LIN {X 0,Y 394.141,Z 720.215,A -85,B 0,C 180,E1 -9307.32,E2 -9307.32} C_VEL
LIN {X 0,Y 395.214,Z 710.247,A -85,B 0,C 180,E1 -9309.27,E2 -9309.27} C_VEL
LIN {X 0,Y 396.4,Z 699.307,A -85,B 0,C 180,E1 -9310.978,E2 -9310.978} C_VEL
LIN {X 0,Y 397.775,Z 685.884,A -85,B 0,C 180,E1 -9312.64,E2 -9312.64} C_VEL
LIN {X 0,Y 399.025,Z 672.379,A -85,B 0,C 180,E1 -9313.952,E2 -9313.952} C_VEL
LIN {X 0,Y 400.251,Z 656.946,A -85,B 0,C 180,E1 -9315.107,E2 -9315.107} C_VEL
LIN {X 0,Y 401.169,Z 641.449,A -85,B 0,C 180,E1 -9315.955,E2 -9315.955} C_VEL
LIN {X 0,Y 401.832,Z 624.77,A -85,B 0,C 180,E1 -9316.577,E2 -9316.577} C_VEL
LIN {X 0,Y 402.409,Z 593.858,A -85,B 0,C 180,E1 -9317.193,E2 -9317.193} C_VEL
LIN {X 0,Y 404.148,Z 493.038,A -85,B 0,C 180,E1 -9319.051,E2 -9319.051} C_VEL
LIN {X 0,Y 402.544,Z 478.977,A -85,B 0,C 180,E1 -9319.466,E2 -9319.466} C_VEL
LIN {X 0,Y 404.689,Z 437.04,A -85,B 0,C 180,E1 -9323.279,E2 -9323.279} C_VEL
LIN {X 0,Y 407.087,Z 392.855,A -85,B 0,C 180,E1 -9327.292,E2 -9327.292} C_VEL
LIN {X 0,Y 409.144,Z 348.932,A -85,B 0,C 180,E1 -9331.221,E2 -9331.221} C_VEL
LIN {X 0,Y 409.823,Z 331.006,A -85,B 0,C 180,E1 -9332.855,E2 -9332.855} C_VEL
LIN {X 0,Y 403.97,Z 313.246,A -85,B 0,C 180,E1 -9335.117,E2 -9335.117} C_VEL
LIN {X 0,Y 396.828,Z 295.284,A -85,B 0,C 180,E1 -9337.637,E2 -9337.637} C_VEL
LIN {X 0,Y 393.6,Z 287.76,A -85,B 0,C 180,E1 -9338.814,E2 -9338.814} C_VEL
LIN {X 0,Y 393.563,Z 287.458,A -85,B 0,C 180,E1 -9340.56,E2 -9340.56} C_VEL
LIN {X 0,Y 393.566,Z 287.451,A -85,B 0,C 180,E1 -9344.528,E2 -9344.528} C_VEL
LIN {X 0,Y 393.561,Z 287.464,A -85,B 0,C 180,E1 -9348.57,E2 -9348.57} C_VEL
LIN {X 0,Y 393.57,Z 287.463,A -85,B 0,C 180,E1 -9352.555,E2 -9352.555} C_VEL
LIN {X 0,Y 393.561,Z 287.461,A -85,B 0,C 180,E1 -9356.65,E2 -9356.65} C_VEL
LIN {X 0,Y 393.569,Z 287.456,A -85,B 0,C 180,E1 -9360.727,E2 -9360.727} C_VEL
LIN {X 0,Y 393.564,Z 287.462,A -85,B 0,C 180,E1 -9364.809,E2 -9364.809} C_VEL
LIN {X 0,Y 393.566,Z 287.458,A -85,B 0,C 180,E1 -9368.804,E2 -9368.804} C_VEL
LIN {X 0,Y 393.564,Z 287.456,A -85,B 0,C 180,E1 -9372.769,E2 -9372.769} C_VEL
LIN {X 0,Y 393.562,Z 287.46,A -85,B 0,C 180,E1 -9376.716,E2 -9376.716} C_VEL
LIN {X 0,Y 393.566,Z 287.46,A -85,B 0,C 180,E1 -9380.793,E2 -9380.793} C_VEL
LIN {X 0,Y 393.562,Z 287.459,A -85,B 0,C 180,E1 -9384.783,E2 -9384.783} C_VEL
LIN {X 0,Y 393.572,Z 287.46,A -85,B 0,C 180,E1 -9388.861,E2 -9388.861} C_VEL
LIN {X 0,Y 393.559,Z 287.463,A -85,B 0,C 180,E1 -9392.766,E2 -9392.766} C_VEL
LIN {X 0,Y 393.553,Z 287.462,A -85,B 0,C 180,E1 -9396.658,E2 -9396.658} C_VEL
LIN {X 0,Y 393.55,Z 287.466,A -85,B 0,C 180,E1 -9400.571,E2 -9400.571} C_VEL
LIN {X 0,Y 393.582,Z 287.73,A -85,B 0,C 180,E1 -9402.449,E2 -9402.449} C_VEL
LIN {X 0,Y 402.202,Z 308.042,A -85,B 0,C 180,E1 -9405.925,E2 -9405.925} C_VEL
LIN {X 0,Y 406.944,Z 319.226,A -85,B 0,C 180,E1 -9407.641,E2 -9407.641} C_VEL
LIN {X 0,Y 422.36,Z 346.857,A -85,B 0,C 180,E1 -9409.922,E2 -9409.922} C_VEL
LIN {X 0,Y 422.986,Z 349.882,A -85,B 0,C 180,E1 -9410.056,E2 -9410.056} C_VEL
LIN {X 0,Y 415.677,Z 539.395,A -85,B 0,C 180,E1 -9413.938,E2 -9413.938} C_VEL
LIN {X 0,Y 414.165,Z 578.769,A -85,B 0,C 180,E1 -9414.777,E2 -9414.777} C_VEL
LIN {X 0,Y 412.749,Z 599.725,A -85,B 0,C 180,E1 -9415.461,E2 -9415.461} C_VEL
LIN {X 0,Y 410.909,Z 620.31,A -85,B 0,C 180,E1 -9416.39,E2 -9416.39} C_VEL
LIN {X 0,Y 408.749,Z 640.92,A -85,B 0,C 180,E1 -9417.61,E2 -9417.61} C_VEL
LIN {X 0,Y 406.395,Z 660.376,A -85,B 0,C 180,E1 -9419.058,E2 -9419.058} C_VEL
LIN {X 0,Y 403.973,Z 678.786,A -85,B 0,C 180,E1 -9420.739,E2 -9420.739} C_VEL
LIN {X 0,Y 401.555,Z 696.152,A -85,B 0,C 180,E1 -9422.654,E2 -9422.654} C_VEL
LIN {X 0,Y 399.377,Z 711.376,A -85,B 0,C 180,E1 -9424.659,E2 -9424.659} C_VEL
LIN {X 0,Y 397.371,Z 725.681,A -85,B 0,C 180,E1 -9426.89,E2 -9426.89} C_VEL
LIN {X 0,Y 395.647,Z 738.602,A -85,B 0,C 180,E1 -9429.282,E2 -9429.282} C_VEL
LIN {X 0,Y 394.254,Z 750.119,A -85,B 0,C 180,E1 -9431.826,E2 -9431.826} C_VEL
LIN {X 0,Y 393.264,Z 759.694,A -85,B 0,C 180,E1 -9434.367,E2 -9434.367} C_VEL
LIN {X 0,Y 392.539,Z 768.289,A -85,B 0,C 180,E1 -9437.199,E2 -9437.199} C_VEL
LIN {X 0,Y 392.165,Z 774.955,A -85,B 0,C 180,E1 -9440.018,E2 -9440.018} C_VEL
LIN {X 0,Y 392.007,Z 779.883,A -85,B 0,C 180,E1 -9442.831,E2 -9442.831} C_VEL
LIN {X 0,Y 391.988,Z 783.143,A -85,B 0,C 180,E1 -9445.613,E2 -9445.613} C_VEL
LIN {X 0,Y 391.999,Z 784.826,A -85,B 0,C 180,E1 -9448.394,E2 -9448.394} C_VEL
LIN {X 0,Y 392.011,Z 784.855,A -85,B 0,C 180,E1 -9451.072,E2 -9451.072} C_VEL
LIN {X 0,Y 392.001,Z 783.287,A -85,B 0,C 180,E1 -9453.95,E2 -9453.95} C_VEL
LIN {X 0,Y 392.02,Z 780.159,A -85,B 0,C 180,E1 -9456.739,E2 -9456.739} C_VEL
LIN {X 0,Y 392.132,Z 775.337,A -85,B 0,C 180,E1 -9459.542,E2 -9459.542} C_VEL
LIN {X 0,Y 392.433,Z 769.064,A -85,B 0,C 180,E1 -9462.21,E2 -9462.21} C_VEL
LIN {X 0,Y 393.049,Z 760.59,A -85,B 0,C 180,E1 -9465.04,E2 -9465.04} C_VEL
LIN {X 0,Y 393.982,Z 750.577,A -85,B 0,C 180,E1 -9467.732,E2 -9467.732} C_VEL
LIN {X 0,Y 395.262,Z 739.097,A -85,B 0,C 180,E1 -9470.278,E2 -9470.278} C_VEL
LIN {X 0,Y 396.852,Z 726.19,A -85,B 0,C 180,E1 -9472.675,E2 -9472.675} C_VEL
LIN {X 0,Y 398.795,Z 711.301,A -85,B 0,C 180,E1 -9474.992,E2 -9474.992} C_VEL
LIN {X 0,Y 401.008,Z 694.704,A -85,B 0,C 180,E1 -9477.149,E2 -9477.149} C_VEL
LIN {X 0,Y 403.385,Z 676.518,A -85,B 0,C 180,E1 -9479.116,E2 -9479.116} C_VEL
LIN {X 0,Y 405.775,Z 657.251,A -85,B 0,C 180,E1 -9480.834,E2 -9480.834} C_VEL
LIN {X 0,Y 408.122,Z 636.959,A -85,B 0,C 180,E1 -9482.306,E2 -9482.306} C_VEL
LIN {X 0,Y 410.253,Z 616.233,A -85,B 0,C 180,E1 -9483.507,E2 -9483.507} C_VEL
LIN {X 0,Y 412.2,Z 594.587,A -85,B 0,C 180,E1 -9484.469,E2 -9484.469} C_VEL
LIN {X 0,Y 413.812,Z 572.25,A -85,B 0,C 180,E1 -9485.184,E2 -9485.184} C_VEL
LIN {X 0,Y 418.128,Z 493.872,A -85,B 0,C 180,E1 -9487.09,E2 -9487.09} C_VEL
LIN {X 0,Y 423.367,Z 428.006,A -85,B 0,C 180,E1 -9488.865,E2 -9488.865} C_VEL
LIN {X 0,Y 430.317,Z 363.895,A -85,B 0,C 180,E1 -9490.73,E2 -9490.73} C_VEL
LIN {X 0,Y 431.806,Z 351.842,A -85,B 0,C 180,E1 -9491.098,E2 -9491.098} C_VEL
LIN {X 0,Y 429.203,Z 345.73,A -85,B 0,C 180,E1 -9492.25,E2 -9492.25} C_VEL
LIN {X 0,Y 426.845,Z 341.145,A -85,B 0,C 180,E1 -9493.567,E2 -9493.567} C_VEL
LIN {X 0,Y 424.814,Z 337.789,A -85,B 0,C 180,E1 -9495.493,E2 -9495.493} C_VEL
LIN {X 0,Y 424.298,Z 337.772,A -85,B 0,C 180,E1 -9496.734,E2 -9496.734} C_VEL
LIN {X 0,Y 424.813,Z 340.3,A -85,B 0,C 180,E1 -9498.662,E2 -9498.662} C_VEL
LIN {X 0,Y 426.33,Z 344.624,A -85,B 0,C 180,E1 -9500.189,E2 -9500.189} C_VEL
LIN {X 0,Y 428.359,Z 350.001,A -85,B 0,C 180,E1 -9501.494,E2 -9501.494} C_VEL
LIN {X 0,Y 429.496,Z 353.537,A -85,B 0,C 180,E1 -9502.122,E2 -9502.122} C_VEL
LIN {X 0,Y 429.664,Z 372.072,A -85,B 0,C 180,E1 -9503.417,E2 -9503.417} C_VEL
LIN {X 0,Y 429.502,Z 378.771,A -85,B 0,C 180,E1 -9503.782,E2 -9503.782} C_VEL
LIN {X 0,Y 420.852,Z 453.997,A -85,B 0,C 180,E1 -9506.036,E2 -9506.036} C_VEL
LIN {X 0,Y 414.952,Z 523.412,A -85,B 0,C 180,E1 -9508.016,E2 -9508.016} C_VEL
LIN {X 0,Y 411.775,Z 569.755,A -85,B 0,C 180,E1 -9509.309,E2 -9509.309} C_VEL
LIN {X 0,Y 410.048,Z 589.973,A -85,B 0,C 180,E1 -9510.13,E2 -9510.13} C_VEL
LIN {X 0,Y 408.054,Z 609.913,A -85,B 0,C 180,E1 -9511.208,E2 -9511.208} C_VEL
LIN {X 0,Y 405.951,Z 628.582,A -85,B 0,C 180,E1 -9512.496,E2 -9512.496} C_VEL
LIN {X 0,Y 403.72,Z 646.478,A -85,B 0,C 180,E1 -9514.03,E2 -9514.03} C_VEL
LIN {X 0,Y 401.544,Z 662.795,A -85,B 0,C 180,E1 -9515.742,E2 -9515.742} C_VEL
LIN {X 0,Y 399.466,Z 677.763,A -85,B 0,C 180,E1 -9517.639,E2 -9517.639} C_VEL
LIN {X 0,Y 397.58,Z 691.237,A -85,B 0,C 180,E1 -9519.693,E2 -9519.693} C_VEL
LIN {X 0,Y 395.933,Z 703.264,A -85,B 0,C 180,E1 -9521.904,E2 -9521.904} C_VEL
LIN {X 0,Y 394.567,Z 713.847,A -85,B 0,C 180,E1 -9524.268,E2 -9524.268} C_VEL
LIN {X 0,Y 393.512,Z 722.946,A -85,B 0,C 180,E1 -9526.781,E2 -9526.781} C_VEL
LIN {X 0,Y 392.803,Z 730.143,A -85,B 0,C 180,E1 -9529.292,E2 -9529.292} C_VEL
LIN {X 0,Y 392.356,Z 735.897,A -85,B 0,C 180,E1 -9531.943,E2 -9531.943} C_VEL
LIN {X 0,Y 392.136,Z 739.907,A -85,B 0,C 180,E1 -9534.587,E2 -9534.587} C_VEL
LIN {X 0,Y 392.039,Z 742.339,A -85,B 0,C 180,E1 -9537.369,E2 -9537.369} C_VEL
LIN {X 0,Y 392.022,Z 743.022,A -85,B 0,C 180,E1 -9540.001,E2 -9540.001} C_VEL
LIN {X 0,Y 392.027,Z 742.021,A -85,B 0,C 180,E1 -9542.778,E2 -9542.778} C_VEL
LIN {X 0,Y 392.1,Z 739.253,A -85,B 0,C 180,E1 -9545.561,E2 -9545.561} C_VEL
LIN {X 0,Y 392.314,Z 734.637,A -85,B 0,C 180,E1 -9548.354,E2 -9548.354} C_VEL
LIN {X 0,Y 392.742,Z 728.456,A -85,B 0,C 180,E1 -9551.008,E2 -9551.008} C_VEL
LIN {X 0,Y 393.485,Z 720.325,A -85,B 0,C 180,E1 -9553.67,E2 -9553.67} C_VEL
LIN {X 0,Y 394.55,Z 710.631,A -85,B 0,C 180,E1 -9556.187,E2 -9556.187} C_VEL
LIN {X 0,Y 395.927,Z 699.422,A -85,B 0,C 180,E1 -9558.554,E2 -9558.554} C_VEL
LIN {X 0,Y 397.59,Z 686.704,A -85,B 0,C 180,E1 -9560.769,E2 -9560.769} C_VEL
LIN {X 0,Y 399.492,Z 672.419,A -85,B 0,C 180,E1 -9562.827,E2 -9562.827} C_VEL
LIN {X 0,Y 401.465,Z 657.392,A -85,B 0,C 180,E1 -9564.625,E2 -9564.625} C_VEL
LIN {X 0,Y 403.508,Z 640.935,A -85,B 0,C 180,E1 -9566.252,E2 -9566.252} C_VEL
LIN {X 0,Y 405.56,Z 622.985,A -85,B 0,C 180,E1 -9567.693,E2 -9567.693} C_VEL
LIN {X 0,Y 407.476,Z 603.872,A -85,B 0,C 180,E1 -9568.908,E2 -9568.908} C_VEL
LIN {X 0,Y 409.102,Z 584.185,A -85,B 0,C 180,E1 -9569.862,E2 -9569.862} C_VEL
LIN {X 0,Y 410.384,Z 564.626,A -85,B 0,C 180,E1 -9570.537,E2 -9570.537} C_VEL
LIN {X 0,Y 411.678,Z 531.02,A -85,B 0,C 180,E1 -9571.28,E2 -9571.28} C_VEL
LIN {X 0,Y 417.674,Z 373.67,A -85,B 0,C 180,E1 -9574.608,E2 -9574.608} C_VEL
LIN {X 0,Y 412.809,Z 339.814,A -85,B 0,C 180,E1 -9575.949,E2 -9575.949} C_VEL
LIN {X 0,Y 412.541,Z 337.856,A -85,B 0,C 180,E1 -9576.187,E2 -9576.187} C_VEL
LIN {X 0,Y 406.059,Z 319.468,A -85,B 0,C 180,E1 -9579.024,E2 -9579.024} C_VEL
LIN {X 0,Y 398.94,Z 301.069,A -85,B 0,C 180,E1 -9582.108,E2 -9582.108} C_VEL
LIN {X 0,Y 393.582,Z 287.659,A -85,B 0,C 180,E1 -9584.556,E2 -9584.556} C_VEL
LIN {X 0,Y 393.563,Z 287.462,A -85,B 0,C 180,E1 -9588.544,E2 -9588.544} C_VEL
LIN {X 0,Y 393.56,Z 287.462,A -85,B 0,C 180,E1 -9592.435,E2 -9592.435} C_VEL
LIN {X 0,Y 393.564,Z 287.463,A -85,B 0,C 180,E1 -9596.44,E2 -9596.44} C_VEL
LIN {X 0,Y 393.559,Z 287.441,A -85,B 0,C 180,E1 -9600.469,E2 -9600.469} C_VEL
LIN {X 0,Y 393.552,Z 287.446,A -85,B 0,C 180,E1 -9604.412,E2 -9604.412} C_VEL
LIN {X 0,Y 393.548,Z 287.449,A -85,B 0,C 180,E1 -9608.382,E2 -9608.382} C_VEL
LIN {X 0,Y 393.536,Z 287.554,A -85,B 0,C 180,E1 -9611.174,E2 -9611.174} C_VEL
LIN {X 0,Y 393.987,Z 289.28,A -85,B 0,C 180,E1 -9611.503,E2 -9611.503} C_VEL
LIN {X 0,Y 401.135,Z 306.789,A -85,B 0,C 180,E1 -9614.011,E2 -9614.011} C_VEL
LIN {X 0,Y 407.641,Z 325.401,A -85,B 0,C 180,E1 -9616.467,E2 -9616.467} C_VEL
LIN {X 0,Y 407.824,Z 328.938,A -85,B 0,C 180,E1 -9616.828,E2 -9616.828} C_VEL
LIN {X 0,Y 406.05,Z 334.761,A -85,B 0,C 180,E1 -9617.234,E2 -9617.234} C_VEL
LIN {X 0,Y 402.635,Z 343.48,A -85,B 0,C 180,E1 -9617.778,E2 -9617.778} C_VEL
LIN {X 0,Y 402.207,Z 346.122,A -85,B 0,C 180,E1 -9617.999,E2 -9617.999} C_VEL
LIN {X 0,Y 399.838,Z 387.755,A -85,B 0,C 180,E1 -9621.876,E2 -9621.876} C_VEL
LIN {X 0,Y 397.374,Z 430.242,A -85,B 0,C 180,E1 -9625.814,E2 -9625.814} C_VEL
LIN {X 0,Y 394.991,Z 472.14,A -85,B 0,C 180,E1 -9629.708,E2 -9629.708} C_VEL
LIN {X 0,Y 394.7,Z 479.497,A -85,B 0,C 180,E1 -9630.357,E2 -9630.357} C_VEL
LIN {X 0,Y 396.483,Z 496.869,A -85,B 0,C 180,E1 -9630.818,E2 -9630.818} C_VEL
LIN {X 0,Y 394.065,Z 622.743,A -85,B 0,C 180,E1 -9633.176,E2 -9633.176} C_VEL
LIN {X 0,Y 393.45,Z 638.836,A -85,B 0,C 180,E1 -9633.746,E2 -9633.746} C_VEL
LIN {X 0,Y 392.507,Z 654.948,A -85,B 0,C 180,E1 -9634.601,E2 -9634.601} C_VEL
LIN {X 0,Y 391.39,Z 669.303,A -85,B 0,C 180,E1 -9635.643,E2 -9635.643} C_VEL
LIN {X 0,Y 390.069,Z 683.635,A -85,B 0,C 180,E1 -9636.992,E2 -9636.992} C_VEL
LIN {X 0,Y 388.772,Z 696.257,A -85,B 0,C 180,E1 -9638.502,E2 -9638.502} C_VEL
LIN {X 0,Y 387.5,Z 707.934,A -85,B 0,C 180,E1 -9640.254,E2 -9640.254} C_VEL
LIN {X 0,Y 386.423,Z 717.792,A -85,B 0,C 180,E1 -9642.096,E2 -9642.096} C_VEL
LIN {X 0,Y 385.467,Z 726.899,A -85,B 0,C 180,E1 -9644.264,E2 -9644.264} C_VEL
LIN {X 0,Y 384.8,Z 734.119,A -85,B 0,C 180,E1 -9646.5,E2 -9646.5} C_VEL
LIN {X 0,Y 384.362,Z 739.874,A -85,B 0,C 180,E1 -9648.974,E2 -9648.974} C_VEL
LIN {X 0,Y 384.158,Z 743.496,A -85,B 0,C 180,E1 -9651.368,E2 -9651.368} C_VEL
LIN {X 0,Y 384.083,Z 745.361,A -85,B 0,C 180,E1 -9653.795,E2 -9653.795} C_VEL
LIN {X 0,Y 384.087,Z 745.527,A -85,B 0,C 180,E1 -9656.098,E2 -9656.098} C_VEL
LIN {X 0,Y 384.166,Z 743.839,A -85,B 0,C 180,E1 -9658.611,E2 -9658.611} C_VEL
LIN {X 0,Y 384.38,Z 740.5,A -85,B 0,C 180,E1 -9660.998,E2 -9660.998} C_VEL
LIN {X 0,Y 384.766,Z 735.571,A -85,B 0,C 180,E1 -9663.249,E2 -9663.249} C_VEL
LIN {X 0,Y 385.43,Z 728.74,A -85,B 0,C 180,E1 -9665.524,E2 -9665.524} C_VEL
LIN {X 0,Y 386.342,Z 720.344,A -85,B 0,C 180,E1 -9667.643,E2 -9667.643} C_VEL
LIN {X 0,Y 387.506,Z 710.223,A -85,B 0,C 180,E1 -9669.649,E2 -9669.649} C_VEL
LIN {X 0,Y 388.761,Z 699.273,A -85,B 0,C 180,E1 -9671.372,E2 -9671.372} C_VEL
LIN {X 0,Y 390.138,Z 686.536,A -85,B 0,C 180,E1 -9672.975,E2 -9672.975} C_VEL
LIN {X 0,Y 391.426,Z 673.431,A -85,B 0,C 180,E1 -9674.284,E2 -9674.284} C_VEL
LIN {X 0,Y 392.715,Z 658.035,A -85,B 0,C 180,E1 -9675.467,E2 -9675.467} C_VEL
LIN {X 0,Y 393.695,Z 642.674,A -85,B 0,C 180,E1 -9676.34,E2 -9676.34} C_VEL
LIN {X 0,Y 394.411,Z 625.713,A -85,B 0,C 180,E1 -9676.993,E2 -9676.993} C_VEL
LIN {X 0,Y 394.914,Z 601.292,A -85,B 0,C 180,E1 -9677.508,E2 -9677.508} C_VEL
LIN {X 0,Y 396.897,Z 494.063,A -85,B 0,C 180,E1 -9679.516,E2 -9679.516} C_VEL
LIN {X 0,Y 395.229,Z 479.296,A -85,B 0,C 180,E1 -9679.968,E2 -9679.968} C_VEL
LIN {X 0,Y 397.566,Z 436.543,A -85,B 0,C 180,E1 -9683.895,E2 -9683.895} C_VEL
LIN {X 0,Y 399.816,Z 396.458,A -85,B 0,C 180,E1 -9687.559,E2 -9687.559} C_VEL
LIN {X 0,Y 401.861,Z 357.064,A -85,B 0,C 180,E1 -9691.138,E2 -9691.138} C_VEL
LIN {X 0,Y 402.887,Z 334.115,A -85,B 0,C 180,E1 -9693.228,E2 -9693.228} C_VEL
LIN {X 0,Y 397.283,Z 316.981,A -85,B 0,C 180,E1 -9695.464,E2 -9695.464} C_VEL
LIN {X 0,Y 390.583,Z 299.994,A -85,B 0,C 180,E1 -9697.894,E2 -9697.894} C_VEL
LIN {X 0,Y 386.577,Z 291.412,A -85,B 0,C 180,E1 -9699.246,E2 -9699.246} C_VEL
LIN {X 0,Y 385.632,Z 288.744,A -85,B 0,C 180,E1 -9699.709,E2 -9699.709} C_VEL
LIN {X 0,Y 385.591,Z 288.444,A -85,B 0,C 180,E1 -9701.713,E2 -9701.713} C_VEL
LIN {X 0,Y 385.59,Z 288.452,A -85,B 0,C 180,E1 -9705.738,E2 -9705.738} C_VEL
LIN {X 0,Y 385.591,Z 288.453,A -85,B 0,C 180,E1 -9709.693,E2 -9709.693} C_VEL
LIN {X 0,Y 385.59,Z 288.45,A -85,B 0,C 180,E1 -9713.747,E2 -9713.747} C_VEL
LIN {X 0,Y 385.59,Z 288.455,A -85,B 0,C 180,E1 -9717.77,E2 -9717.77} C_VEL
LIN {X 0,Y 385.591,Z 288.45,A -85,B 0,C 180,E1 -9721.783,E2 -9721.783} C_VEL
LIN {X 0,Y 385.592,Z 288.454,A -85,B 0,C 180,E1 -9725.804,E2 -9725.804} C_VEL
LIN {X 0,Y 385.593,Z 288.446,A -85,B 0,C 180,E1 -9729.854,E2 -9729.854} C_VEL
LIN {X 0,Y 385.594,Z 288.452,A -85,B 0,C 180,E1 -9733.954,E2 -9733.954} C_VEL
LIN {X 0,Y 385.596,Z 288.453,A -85,B 0,C 180,E1 -9737.973,E2 -9737.973} C_VEL
LIN {X 0,Y 385.593,Z 288.447,A -85,B 0,C 180,E1 -9741.925,E2 -9741.925} C_VEL
LIN {X 0,Y 385.597,Z 288.453,A -85,B 0,C 180,E1 -9745.99,E2 -9745.99} C_VEL
LIN {X 0,Y 385.6,Z 288.449,A -85,B 0,C 180,E1 -9750.029,E2 -9750.029} C_VEL
LIN {X 0,Y 385.6,Z 288.45,A -85,B 0,C 180,E1 -9754.061,E2 -9754.061} C_VEL
LIN {X 0,Y 385.601,Z 288.45,A -85,B 0,C 180,E1 -9758.106,E2 -9758.106} C_VEL
LIN {X 0,Y 385.659,Z 288.721,A -85,B 0,C 180,E1 -9761.528,E2 -9761.528} C_VEL
LIN {X 0,Y 388.596,Z 295.735,A -85,B 0,C 180,E1 -9762.839,E2 -9762.839} C_VEL
LIN {X 0,Y 397.618,Z 316.933,A -85,B 0,C 180,E1 -9766.403,E2 -9766.403} C_VEL
LIN {X 0,Y 398.948,Z 319.876,A -85,B 0,C 180,E1 -9766.802,E2 -9766.802} C_VEL
LIN {X 0,Y 414.538,Z 347.5,A -85,B 0,C 180,E1 -9769.179,E2 -9769.179} C_VEL
LIN {X 0,Y 416.358,Z 351.397,A -85,B 0,C 180,E1 -9769.461,E2 -9769.461} C_VEL
LIN {X 0,Y 408.437,Z 546.701,A -85,B 0,C 180,E1 -9773.542,E2 -9773.542} C_VEL
LIN {X 0,Y 407.015,Z 580.064,A -85,B 0,C 180,E1 -9774.29,E2 -9774.29} C_VEL
LIN {X 0,Y 405.492,Z 601.047,A -85,B 0,C 180,E1 -9775.006,E2 -9775.006} C_VEL
LIN {X 0,Y 403.586,Z 621.322,A -85,B 0,C 180,E1 -9775.953,E2 -9775.953} C_VEL
LIN {X 0,Y 401.48,Z 640.647,A -85,B 0,C 180,E1 -9777.12,E2 -9777.12} C_VEL
LIN {X 0,Y 399.03,Z 660.122,A -85,B 0,C 180,E1 -9778.59,E2 -9778.59} C_VEL
LIN {X 0,Y 396.51,Z 678.559,A -85,B 0,C 180,E1 -9780.299,E2 -9780.299} C_VEL
LIN {X 0,Y 394.072,Z 695.297,A -85,B 0,C 180,E1 -9782.172,E2 -9782.172} C_VEL
LIN {X 0,Y 391.716,Z 711.133,A -85,B 0,C 180,E1 -9784.285,E2 -9784.285} C_VEL
LIN {X 0,Y 389.616,Z 725.484,A -85,B 0,C 180,E1 -9786.563,E2 -9786.563} C_VEL
LIN {X 0,Y 387.808,Z 738.415,A -85,B 0,C 180,E1 -9789.002,E2 -9789.002} C_VEL
LIN {X 0,Y 386.351,Z 749.923,A -85,B 0,C 180,E1 -9791.597,E2 -9791.597} C_VEL
LIN {X 0,Y 385.269,Z 759.915,A -85,B 0,C 180,E1 -9794.327,E2 -9794.327} C_VEL
LIN {X 0,Y 384.53,Z 768.479,A -85,B 0,C 180,E1 -9797.233,E2 -9797.233} C_VEL
LIN {X 0,Y 384.157,Z 775.03,A -85,B 0,C 180,E1 -9800.11,E2 -9800.11} C_VEL
LIN {X 0,Y 384.012,Z 779.583,A -85,B 0,C 180,E1 -9802.822,E2 -9802.822} C_VEL
LIN {X 0,Y 383.999,Z 782.86,A -85,B 0,C 180,E1 -9805.751,E2 -9805.751} C_VEL
LIN {X 0,Y 384.011,Z 784.423,A -85,B 0,C 180,E1 -9808.51,E2 -9808.51} C_VEL
LIN {X 0,Y 384.02,Z 784.396,A -85,B 0,C 180,E1 -9811.195,E2 -9811.195} C_VEL
LIN {X 0,Y 384.009,Z 782.846,A -85,B 0,C 180,E1 -9814.033,E2 -9814.033} C_VEL
LIN {X 0,Y 384.024,Z 779.703,A -85,B 0,C 180,E1 -9816.88,E2 -9816.88} C_VEL
LIN {X 0,Y 384.151,Z 774.855,A -85,B 0,C 180,E1 -9819.742,E2 -9819.742} C_VEL
LIN {X 0,Y 384.471,Z 768.554,A -85,B 0,C 180,E1 -9822.467,E2 -9822.467} C_VEL
LIN {X 0,Y 385.142,Z 760.046,A -85,B 0,C 180,E1 -9825.357,E2 -9825.357} C_VEL
LIN {X 0,Y 386.17,Z 749.788,A -85,B 0,C 180,E1 -9828.155,E2 -9828.155} C_VEL
LIN {X 0,Y 387.524,Z 738.476,A -85,B 0,C 180,E1 -9830.702,E2 -9830.702} C_VEL
LIN {X 0,Y 389.231,Z 725.53,A -85,B 0,C 180,E1 -9833.144,E2 -9833.144} C_VEL
LIN {X 0,Y 391.309,Z 710.607,A -85,B 0,C 180,E1 -9835.504,E2 -9835.504} C_VEL
LIN {X 0,Y 393.671,Z 693.985,A -85,B 0,C 180,E1 -9837.698,E2 -9837.698} C_VEL
LIN {X 0,Y 396.149,Z 676.253,A -85,B 0,C 180,E1 -9839.651,E2 -9839.651} C_VEL
LIN {X 0,Y 398.765,Z 656.587,A -85,B 0,C 180,E1 -9841.437,E2 -9841.437} C_VEL
LIN {X 0,Y 401.223,Z 636.704,A -85,B 0,C 180,E1 -9842.907,E2 -9842.907} C_VEL
LIN {X 0,Y 403.581,Z 615.51,A -85,B 0,C 180,E1 -9844.16,E2 -9844.16} C_VEL
LIN {X 0,Y 405.687,Z 593.804,A -85,B 0,C 180,E1 -9845.146,E2 -9845.146} C_VEL
LIN {X 0,Y 407.476,Z 571.241,A -85,B 0,C 180,E1 -9845.885,E2 -9845.885} C_VEL
LIN {X 0,Y 412.132,Z 497.627,A -85,B 0,C 180,E1 -9847.767,E2 -9847.767} C_VEL
LIN {X 0,Y 417.762,Z 434.94,A -85,B 0,C 180,E1 -9849.532,E2 -9849.532} C_VEL
LIN {X 0,Y 425.447,Z 371.518,A -85,B 0,C 180,E1 -9851.446,E2 -9851.446} C_VEL
LIN {X 0,Y 427.584,Z 355.86,A -85,B 0,C 180,E1 -9851.961,E2 -9851.961} C_VEL
LIN {X 0,Y 425.739,Z 351.406,A -85,B 0,C 180,E1 -9852.949,E2 -9852.949} C_VEL
LIN {X 0,Y 424.157,Z 348.165,A -85,B 0,C 180,E1 -9854.031,E2 -9854.031} C_VEL
LIN {X 0,Y 422.802,Z 345.516,A -85,B 0,C 180,E1 -9855.577,E2 -9855.577} C_VEL
LIN {X 0,Y 422.342,Z 345.513,A -85,B 0,C 180,E1 -9856.643,E2 -9856.643} C_VEL
LIN {X 0,Y 422.646,Z 347.936,A -85,B 0,C 180,E1 -9858.472,E2 -9858.472} C_VEL
LIN {X 0,Y 423.852,Z 352.079,A -85,B 0,C 180,E1 -9859.941,E2 -9859.941} C_VEL
LIN {X 0,Y 425.435,Z 357.078,A -85,B 0,C 180,E1 -9861.134,E2 -9861.134} C_VEL
LIN {X 0,Y 425.847,Z 358.986,A -85,B 0,C 180,E1 -9861.443,E2 -9861.443} C_VEL
LIN {X 0,Y 425.438,Z 376.705,A -85,B 0,C 180,E1 -9862.698,E2 -9862.698} C_VEL
LIN {X 0,Y 425.151,Z 380.959,A -85,B 0,C 180,E1 -9862.915,E2 -9862.915} C_VEL
LIN {X 0,Y 415.891,Z 452.689,A -85,B 0,C 180,E1 -9865.145,E2 -9865.145} C_VEL
LIN {X 0,Y 409.352,Z 519.498,A -85,B 0,C 180,E1 -9867.151,E2 -9867.151} C_VEL
LIN {X 0,Y 405.386,Z 570.426,A -85,B 0,C 180,E1 -9868.64,E2 -9868.64} C_VEL
LIN {X 0,Y 403.425,Z 591.228,A -85,B 0,C 180,E1 -9869.521,E2 -9869.521} C_VEL
LIN {X 0,Y 401.306,Z 610.6,A -85,B 0,C 180,E1 -9870.605,E2 -9870.605} C_VEL
LIN {X 0,Y 398.96,Z 629.842,A -85,B 0,C 180,E1 -9871.972,E2 -9871.972} C_VEL
LIN {X 0,Y 396.521,Z 647.903,A -85,B 0,C 180,E1 -9873.573,E2 -9873.573} C_VEL
LIN {X 0,Y 394.184,Z 664.215,A -85,B 0,C 180,E1 -9875.339,E2 -9875.339} C_VEL
LIN {X 0,Y 391.906,Z 679.493,A -85,B 0,C 180,E1 -9877.342,E2 -9877.342} C_VEL
LIN {X 0,Y 389.92,Z 692.735,A -85,B 0,C 180,E1 -9879.433,E2 -9879.433} C_VEL
LIN {X 0,Y 388.182,Z 704.572,A -85,B 0,C 180,E1 -9881.685,E2 -9881.685} C_VEL
LIN {X 0,Y 386.73,Z 715.054,A -85,B 0,C 180,E1 -9884.11,E2 -9884.11} C_VEL
LIN {X 0,Y 385.62,Z 723.955,A -85,B 0,C 180,E1 -9886.658,E2 -9886.658} C_VEL
LIN {X 0,Y 384.866,Z 731.025,A -85,B 0,C 180,E1 -9889.22,E2 -9889.22} C_VEL
LIN {X 0,Y 384.39,Z 736.661,A -85,B 0,C 180,E1 -9891.926,E2 -9891.926} C_VEL
LIN {X 0,Y 384.156,Z 740.555,A -85,B 0,C 180,E1 -9894.624,E2 -9894.624} C_VEL
LIN {X 0,Y 384.055,Z 742.806,A -85,B 0,C 180,E1 -9897.315,E2 -9897.315} C_VEL
LIN {X 0,Y 384.034,Z 743.462,A -85,B 0,C 180,E1 -9900.001,E2 -9900.001} C_VEL
LIN {X 0,Y 384.039,Z 742.418,A -85,B 0,C 180,E1 -9902.836,E2 -9902.836} C_VEL
LIN {X 0,Y 384.119,Z 739.593,A -85,B 0,C 180,E1 -9905.677,E2 -9905.677} C_VEL
LIN {X 0,Y 384.335,Z 735.21,A -85,B 0,C 180,E1 -9908.378,E2 -9908.378} C_VEL
LIN {X 0,Y 384.782,Z 729.053,A -85,B 0,C 180,E1 -9911.087,E2 -9911.087} C_VEL
LIN {X 0,Y 385.56,Z 720.955,A -85,B 0,C 180,E1 -9913.803,E2 -9913.803} C_VEL
LIN {X 0,Y 386.687,Z 711.151,A -85,B 0,C 180,E1 -9916.401,E2 -9916.401} C_VEL
LIN {X 0,Y 388.11,Z 700.088,A -85,B 0,C 180,E1 -9918.786,E2 -9918.786} C_VEL
LIN {X 0,Y 389.844,Z 687.4,A -85,B 0,C 180,E1 -9921.044,E2 -9921.044} C_VEL
LIN {X 0,Y 391.826,Z 673.161,A -85,B 0,C 180,E1 -9923.14,E2 -9923.14} C_VEL
LIN {X 0,Y 393.943,Z 657.683,A -85,B 0,C 180,E1 -9925.027,E2 -9925.027} C_VEL
LIN {X 0,Y 396.1,Z 640.996,A -85,B 0,C 180,E1 -9926.701,E2 -9926.701} C_VEL
LIN {X 0,Y 398.237,Z 622.993,A -85,B 0,C 180,E1 -9928.166,E2 -9928.166} C_VEL
LIN {X 0,Y 400.237,Z 603.839,A -85,B 0,C 180,E1 -9929.4,E2 -9929.4} C_VEL
LIN {X 0,Y 401.921,Z 584.234,A -85,B 0,C 180,E1 -9930.363,E2 -9930.363} C_VEL
LIN {X 0,Y 403.261,Z 564.613,A -85,B 0,C 180,E1 -9931.052,E2 -9931.052} C_VEL
LIN {X 0,Y 404.762,Z 527.661,A -85,B 0,C 180,E1 -9931.888,E2 -9931.888} C_VEL
LIN {X 0,Y 410.951,Z 374.818,A -85,B 0,C 180,E1 -9935.2,E2 -9935.2} C_VEL
LIN {X 0,Y 406.023,Z 341.792,A -85,B 0,C 180,E1 -9936.541,E2 -9936.541} C_VEL
LIN {X 0,Y 404.74,Z 338.868,A -85,B 0,C 180,E1 -9936.83,E2 -9936.83} C_VEL
LIN {X 0,Y 398.098,Z 320.346,A -85,B 0,C 180,E1 -9939.775,E2 -9939.775} C_VEL
LIN {X 0,Y 390.871,Z 301.781,A -85,B 0,C 180,E1 -9942.978,E2 -9942.978} C_VEL
LIN {X 0,Y 385.651,Z 288.651,A -85,B 0,C 180,E1 -9945.456,E2 -9945.456} C_VEL
LIN {X 0,Y 385.626,Z 288.452,A -85,B 0,C 180,E1 -9949.438,E2 -9949.438} C_VEL
LIN {X 0,Y 385.621,Z 288.448,A -85,B 0,C 180,E1 -9953.494,E2 -9953.494} C_VEL
LIN {X 0,Y 385.621,Z 288.449,A -85,B 0,C 180,E1 -9957.538,E2 -9957.538} C_VEL
LIN {X 0,Y 385.618,Z 288.434,A -85,B 0,C 180,E1 -9961.521,E2 -9961.521} C_VEL
LIN {X 0,Y 385.609,Z 288.434,A -85,B 0,C 180,E1 -9965.524,E2 -9965.524} C_VEL
LIN {X 0,Y 385.596,Z 288.441,A -85,B 0,C 180,E1 -9969.405,E2 -9969.405} C_VEL
LIN {X 0,Y 385.63,Z 288.664,A -85,B 0,C 180,E1 -9970.458,E2 -9970.458} C_VEL
LIN {X 0,Y 388.127,Z 294.947,A -85,B 0,C 180,E1 -9971.446,E2 -9971.446} C_VEL
LIN {X 0,Y 395.619,Z 313.822,A -85,B 0,C 180,E1 -9974.159,E2 -9974.159} C_VEL
LIN {X 0,Y 402.27,Z 333.616,A -85,B 0,C 180,E1 -9976.78,E2 -9976.78} C_VEL
LIN {X 0,Y 402.753,Z 336.308,A -85,B 0,C 180,E1 -9977.088,E2 -9977.088} C_VEL
LIN {X 0,Y 402.207,Z 346.122,A -85,B 0,C 180,E1 -9977.999,E2 -9977.999} C_VEL
LIN {X 0,Y 400.979,Z 352.785,A -85,B 0,C 180,E1 -9978.539,E2 -9978.539} C_VEL
LIN {X 0,Y 394.437,Z 371.147,A -85,B 0,C 180,E1 -9979.766,E2 -9979.766} C_VEL
LIN {X 0,Y 393.42,Z 376.867,A -85,B 0,C 180,E1 -9980.245,E2 -9980.245} C_VEL
LIN {X 0,Y 390.87,Z 418.201,A -85,B 0,C 180,E1 -9984.126,E2 -9984.126} C_VEL
LIN {X 0,Y 388.343,Z 461.181,A -85,B 0,C 180,E1 -9988.154,E2 -9988.154} C_VEL
LIN {X 0,Y 387.324,Z 479.827,A -85,B 0,C 180,E1 -9989.874,E2 -9989.874} C_VEL
LIN {X 0,Y 389.149,Z 497.663,A -85,B 0,C 180,E1 -9990.36,E2 -9990.36} C_VEL
LIN {X 0,Y 386.608,Z 623.155,A -85,B 0,C 180,E1 -9992.755,E2 -9992.755} C_VEL
LIN {X 0,Y 385.965,Z 639.192,A -85,B 0,C 180,E1 -9993.333,E2 -9993.333} C_VEL
LIN {X 0,Y 384.984,Z 655.233,A -85,B 0,C 180,E1 -9994.199,E2 -9994.199} C_VEL
LIN {X 0,Y 383.849,Z 669.257,A -85,B 0,C 180,E1 -9995.229,E2 -9995.229} C_VEL
LIN {X 0,Y 382.459,Z 683.671,A -85,B 0,C 180,E1 -9996.604,E2 -9996.604} C_VEL
LIN {X 0,Y 381.091,Z 696.381,A -85,B 0,C 180,E1 -9998.143,E2 -9998.143} C_VEL
LIN {X 0,Y 379.695,Z 708.569,A -85,B 0,C 180,E1 -10000.007,E2 -10000.007} C_VEL
LIN {X 0,Y 378.562,Z 718.372,A -85,B 0,C 180,E1 -10001.887,E2 -10001.887} C_VEL
LIN {X 0,Y 377.555,Z 727.448,A -85,B 0,C 180,E1 -10004.099,E2 -10004.099} C_VEL
LIN {X 0,Y 376.862,Z 734.493,A -85,B 0,C 180,E1 -10006.332,E2 -10006.332} C_VEL
LIN {X 0,Y 376.406,Z 740.037,A -85,B 0,C 180,E1 -10008.747,E2 -10008.747} C_VEL
LIN {X 0,Y 376.179,Z 743.765,A -85,B 0,C 180,E1 -10011.189,E2 -10011.189} C_VEL
LIN {X 0,Y 376.095,Z 745.698,A -85,B 0,C 180,E1 -10013.666,E2 -10013.666} C_VEL
LIN {X 0,Y 376.098,Z 745.901,A -85,B 0,C 180,E1 -10016.185,E2 -10016.185} C_VEL
LIN {X 0,Y 376.188,Z 744.18,A -85,B 0,C 180,E1 -10018.753,E2 -10018.753} C_VEL
LIN {X 0,Y 376.427,Z 740.771,A -85,B 0,C 180,E1 -10021.207,E2 -10021.207} C_VEL
LIN {X 0,Y 376.894,Z 735.364,A -85,B 0,C 180,E1 -10023.671,E2 -10023.671} C_VEL
LIN {X 0,Y 377.598,Z 728.744,A -85,B 0,C 180,E1 -10025.876,E2 -10025.876} C_VEL
LIN {X 0,Y 378.619,Z 719.95,A -85,B 0,C 180,E1 -10028.096,E2 -10028.096} C_VEL
LIN {X 0,Y 379.783,Z 710.471,A -85,B 0,C 180,E1 -10029.992,E2 -10029.992} C_VEL
LIN {X 0,Y 381.141,Z 699.241,A -85,B 0,C 180,E1 -10031.781,E2 -10031.781} C_VEL
LIN {X 0,Y 382.607,Z 686.432,A -85,B 0,C 180,E1 -10033.413,E2 -10033.413} C_VEL
LIN {X 0,Y 383.966,Z 673.167,A -85,B 0,C 180,E1 -10034.746,E2 -10034.746} C_VEL
LIN {X 0,Y 385.314,Z 657.803,A -85,B 0,C 180,E1 -10035.937,E2 -10035.937} C_VEL
LIN {X 0,Y 386.332,Z 642.25,A -85,B 0,C 180,E1 -10036.82,E2 -10036.82} C_VEL
LIN {X 0,Y 387.065,Z 625.559,A -85,B 0,C 180,E1 -10037.464,E2 -10037.464} C_VEL
LIN {X 0,Y 387.736,Z 593.398,A -85,B 0,C 180,E1 -10038.128,E2 -10038.128} C_VEL
LIN {X 0,Y 389.648,Z 494.75,A -85,B 0,C 180,E1 -10040.01,E2 -10040.01} C_VEL
LIN {X 0,Y 387.952,Z 480.003,A -85,B 0,C 180,E1 -10040.461,E2 -10040.461} C_VEL
LIN {X 0,Y 390.482,Z 436.326,A -85,B 0,C 180,E1 -10044.511,E2 -10044.511} C_VEL
LIN {X 0,Y 393.042,Z 393.106,A -85,B 0,C 180,E1 -10048.513,E2 -10048.513} C_VEL
LIN {X 0,Y 395.389,Z 349.348,A -85,B 0,C 180,E1 -10052.515,E2 -10052.515} C_VEL
LIN {X 0,Y 396.024,Z 337.35,A -85,B 0,C 180,E1 -10053.617,E2 -10053.617} C_VEL
LIN {X 0,Y 390.695,Z 320.827,A -85,B 0,C 180,E1 -10055.828,E2 -10055.828} C_VEL
LIN {X 0,Y 384.015,Z 303.953,A -85,B 0,C 180,E1 -10058.301,E2 -10058.301} C_VEL
LIN {X 0,Y 378.89,Z 292.803,A -85,B 0,C 180,E1 -10060.097,E2 -10060.097} C_VEL
LIN {X 0,Y 377.731,Z 289.764,A -85,B 0,C 180,E1 -10060.637,E2 -10060.637} C_VEL
LIN {X 0,Y 377.654,Z 289.433,A -85,B 0,C 180,E1 -10061.795,E2 -10061.795} C_VEL
LIN {X 0,Y 377.653,Z 289.441,A -85,B 0,C 180,E1 -10065.745,E2 -10065.745} C_VEL
LIN {X 0,Y 377.653,Z 289.443,A -85,B 0,C 180,E1 -10069.782,E2 -10069.782} C_VEL
LIN {X 0,Y 377.652,Z 289.439,A -85,B 0,C 180,E1 -10073.768,E2 -10073.768} C_VEL
LIN {X 0,Y 377.652,Z 289.442,A -85,B 0,C 180,E1 -10077.875,E2 -10077.875} C_VEL
LIN {X 0,Y 377.653,Z 289.439,A -85,B 0,C 180,E1 -10081.82,E2 -10081.82} C_VEL
LIN {X 0,Y 377.655,Z 289.443,A -85,B 0,C 180,E1 -10085.926,E2 -10085.926} C_VEL
LIN {X 0,Y 377.655,Z 289.435,A -85,B 0,C 180,E1 -10089.988,E2 -10089.988} C_VEL
LIN {X 0,Y 377.658,Z 289.442,A -85,B 0,C 180,E1 -10094.097,E2 -10094.097} C_VEL
LIN {X 0,Y 377.661,Z 289.44,A -85,B 0,C 180,E1 -10098.204,E2 -10098.204} C_VEL
LIN {X 0,Y 377.66,Z 289.436,A -85,B 0,C 180,E1 -10102.246,E2 -10102.246} C_VEL
LIN {X 0,Y 377.662,Z 289.443,A -85,B 0,C 180,E1 -10106.24,E2 -10106.24} C_VEL
LIN {X 0,Y 377.663,Z 289.438,A -85,B 0,C 180,E1 -10110.2,E2 -10110.2} C_VEL
LIN {X 0,Y 377.664,Z 289.439,A -85,B 0,C 180,E1 -10114.326,E2 -10114.326} C_VEL
LIN {X 0,Y 377.666,Z 289.44,A -85,B 0,C 180,E1 -10118.408,E2 -10118.408} C_VEL
LIN {X 0,Y 377.716,Z 289.737,A -85,B 0,C 180,E1 -10120.591,E2 -10120.591} C_VEL
LIN {X 0,Y 386.088,Z 309.298,A -85,B 0,C 180,E1 -10124.157,E2 -10124.157} C_VEL
LIN {X 0,Y 390.517,Z 319.683,A -85,B 0,C 180,E1 -10125.855,E2 -10125.855} C_VEL
LIN {X 0,Y 407.06,Z 348.807,A -85,B 0,C 180,E1 -10128.46,E2 -10128.46} C_VEL
LIN {X 0,Y 409.737,Z 354.251,A -85,B 0,C 180,E1 -10128.87,E2 -10128.87} C_VEL
LIN {X 0,Y 401.571,Z 543.738,A -85,B 0,C 180,E1 -10132.925,E2 -10132.925} C_VEL
LIN {X 0,Y 399.995,Z 579.391,A -85,B 0,C 180,E1 -10133.734,E2 -10133.734} C_VEL
LIN {X 0,Y 398.438,Z 600.282,A -85,B 0,C 180,E1 -10134.453,E2 -10134.453} C_VEL
LIN {X 0,Y 396.573,Z 619.61,A -85,B 0,C 180,E1 -10135.354,E2 -10135.354} C_VEL
LIN {X 0,Y 394.235,Z 640.263,A -85,B 0,C 180,E1 -10136.611,E2 -10136.611} C_VEL
LIN {X 0,Y 391.688,Z 659.766,A -85,B 0,C 180,E1 -10138.105,E2 -10138.105} C_VEL
LIN {X 0,Y 389.061,Z 678.211,A -85,B 0,C 180,E1 -10139.842,E2 -10139.842} C_VEL
LIN {X 0,Y 386.426,Z 695.615,A -85,B 0,C 180,E1 -10141.824,E2 -10141.824} C_VEL
LIN {X 0,Y 384.038,Z 711.023,A -85,B 0,C 180,E1 -10143.925,E2 -10143.925} C_VEL
LIN {X 0,Y 381.869,Z 725.235,A -85,B 0,C 180,E1 -10146.222,E2 -10146.222} C_VEL
LIN {X 0,Y 379.977,Z 738.176,A -85,B 0,C 180,E1 -10148.71,E2 -10148.71} C_VEL
LIN {X 0,Y 378.451,Z 749.682,A -85,B 0,C 180,E1 -10151.359,E2 -10151.359} C_VEL
LIN {X 0,Y 377.326,Z 759.627,A -85,B 0,C 180,E1 -10154.131,E2 -10154.131} C_VEL
LIN {X 0,Y 376.568,Z 767.994,A -85,B 0,C 180,E1 -10157.02,E2 -10157.02} C_VEL
LIN {X 0,Y 376.163,Z 774.767,A -85,B 0,C 180,E1 -10160.053,E2 -10160.053} C_VEL
LIN {X 0,Y 376.018,Z 779.281,A -85,B 0,C 180,E1 -10162.822,E2 -10162.822} C_VEL
LIN {X 0,Y 376.01,Z 782.442,A -85,B 0,C 180,E1 -10165.732,E2 -10165.732} C_VEL
LIN {X 0,Y 376.025,Z 784,A -85,B 0,C 180,E1 -10168.63,E2 -10168.63} C_VEL
LIN {X 0,Y 376.03,Z 783.923,A -85,B 0,C 180,E1 -10171.373,E2 -10171.373} C_VEL
LIN {X 0,Y 376.014,Z 782.237,A -85,B 0,C 180,E1 -10174.321,E2 -10174.321} C_VEL
LIN {X 0,Y 376.027,Z 778.801,A -85,B 0,C 180,E1 -10177.334,E2 -10177.334} C_VEL
LIN {X 0,Y 376.183,Z 774.096,A -85,B 0,C 180,E1 -10180.105,E2 -10180.105} C_VEL
LIN {X 0,Y 376.573,Z 767.289,A -85,B 0,C 180,E1 -10183.045,E2 -10183.045} C_VEL
LIN {X 0,Y 377.294,Z 759.002,A -85,B 0,C 180,E1 -10185.852,E2 -10185.852} C_VEL
LIN {X 0,Y 378.404,Z 748.838,A -85,B 0,C 180,E1 -10188.647,E2 -10188.647} C_VEL
LIN {X 0,Y 380.005,Z 736.395,A -85,B 0,C 180,E1 -10191.454,E2 -10191.454} C_VEL
LIN {X 0,Y 381.94,Z 722.847,A -85,B 0,C 180,E1 -10193.989,E2 -10193.989} C_VEL
LIN {X 0,Y 384.155,Z 708.03,A -85,B 0,C 180,E1 -10196.317,E2 -10196.317} C_VEL
LIN {X 0,Y 386.6,Z 691.972,A -85,B 0,C 180,E1 -10198.438,E2 -10198.438} C_VEL
LIN {X 0,Y 389.239,Z 674.193,A -85,B 0,C 180,E1 -10200.402,E2 -10200.402} C_VEL
LIN {X 0,Y 391.918,Z 655.491,A -85,B 0,C 180,E1 -10202.114,E2 -10202.114} C_VEL
LIN {X 0,Y 394.59,Z 635.283,A -85,B 0,C 180,E1 -10203.627,E2 -10203.627} C_VEL
LIN {X 0,Y 397.071,Z 614.668,A -85,B 0,C 180,E1 -10204.864,E2 -10204.864} C_VEL
LIN {X 0,Y 399.349,Z 593.081,A -85,B 0,C 180,E1 -10205.866,E2 -10205.866} C_VEL
LIN {X 0,Y 401.355,Z 570.136,A -85,B 0,C 180,E1 -10206.637,E2 -10206.637} C_VEL
LIN {X 0,Y 406.419,Z 500.604,A -85,B 0,C 180,E1 -10208.507,E2 -10208.507} C_VEL
LIN {X 0,Y 412.494,Z 440.99,A -85,B 0,C 180,E1 -10210.263,E2 -10210.263} C_VEL
LIN {X 0,Y 420.617,Z 380.86,A -85,B 0,C 180,E1 -10212.141,E2 -10212.141} C_VEL
LIN {X 0,Y 423.847,Z 360.47,A -85,B 0,C 180,E1 -10212.807,E2 -10212.807} C_VEL
LIN {X 0,Y 422.14,Z 356.085,A -85,B 0,C 180,E1 -10214.041,E2 -10214.041} C_VEL
LIN {X 0,Y 420.779,Z 353.237,A -85,B 0,C 180,E1 -10215.685,E2 -10215.685} C_VEL
LIN {X 0,Y 420.316,Z 353.415,A -85,B 0,C 180,E1 -10216.714,E2 -10216.714} C_VEL
LIN {X 0,Y 420.495,Z 355.616,A -85,B 0,C 180,E1 -10218.301,E2 -10218.301} C_VEL
LIN {X 0,Y 421.439,Z 359.627,A -85,B 0,C 180,E1 -10219.699,E2 -10219.699} C_VEL
LIN {X 0,Y 422.49,Z 363.795,A -85,B 0,C 180,E1 -10220.685,E2 -10220.685} C_VEL
LIN {X 0,Y 421.522,Z 380.833,A -85,B 0,C 180,E1 -10221.912,E2 -10221.912} C_VEL
LIN {X 0,Y 411.493,Z 450.143,A -85,B 0,C 180,E1 -10224.161,E2 -10224.161} C_VEL
LIN {X 0,Y 404.087,Z 516.008,A -85,B 0,C 180,E1 -10226.233,E2 -10226.233} C_VEL
LIN {X 0,Y 399.163,Z 571.366,A -85,B 0,C 180,E1 -10227.936,E2 -10227.936} C_VEL
LIN {X 0,Y 397.052,Z 591.572,A -85,B 0,C 180,E1 -10228.824,E2 -10228.824} C_VEL
LIN {X 0,Y 394.706,Z 611.287,A -85,B 0,C 180,E1 -10229.959,E2 -10229.959} C_VEL
LIN {X 0,Y 392.165,Z 630.471,A -85,B 0,C 180,E1 -10231.359,E2 -10231.359} C_VEL
LIN {X 0,Y 389.562,Z 648.351,A -85,B 0,C 180,E1 -10232.981,E2 -10232.981} C_VEL
LIN {X 0,Y 387.063,Z 664.574,A -85,B 0,C 180,E1 -10234.772,E2 -10234.772} C_VEL
LIN {X 0,Y 384.714,Z 679.307,A -85,B 0,C 180,E1 -10236.732,E2 -10236.732} C_VEL
LIN {X 0,Y 382.565,Z 692.626,A -85,B 0,C 180,E1 -10238.859,E2 -10238.859} C_VEL
LIN {X 0,Y 380.677,Z 704.546,A -85,B 0,C 180,E1 -10241.152,E2 -10241.152} C_VEL
LIN {X 0,Y 379.096,Z 715.051,A -85,B 0,C 180,E1 -10243.608,E2 -10243.608} C_VEL
LIN {X 0,Y 377.852,Z 724.092,A -85,B 0,C 180,E1 -10246.223,E2 -10246.223} C_VEL
LIN {X 0,Y 376.99,Z 731.413,A -85,B 0,C 180,E1 -10248.912,E2 -10248.912} C_VEL
LIN {X 0,Y 376.472,Z 736.951,A -85,B 0,C 180,E1 -10251.601,E2 -10251.601} C_VEL
LIN {X 0,Y 376.195,Z 740.911,A -85,B 0,C 180,E1 -10254.357,E2 -10254.357} C_VEL
LIN {X 0,Y 376.078,Z 743.22,A -85,B 0,C 180,E1 -10257.105,E2 -10257.105} C_VEL
LIN {X 0,Y 376.045,Z 743.906,A -85,B 0,C 180,E1 -10259.848,E2 -10259.848} C_VEL
LIN {X 0,Y 376.045,Z 742.986,A -85,B 0,C 180,E1 -10262.591,E2 -10262.591} C_VEL
LIN {X 0,Y 376.115,Z 740.47,A -85,B 0,C 180,E1 -10265.339,E2 -10265.339} C_VEL
LIN {X 0,Y 376.317,Z 736.296,A -85,B 0,C 180,E1 -10268.096,E2 -10268.096} C_VEL
LIN {X 0,Y 376.755,Z 730.362,A -85,B 0,C 180,E1 -10270.861,E2 -10270.861} C_VEL
LIN {X 0,Y 377.502,Z 722.694,A -85,B 0,C 180,E1 -10273.576,E2 -10273.576} C_VEL
LIN {X 0,Y 378.557,Z 713.707,A -85,B 0,C 180,E1 -10276.102,E2 -10276.102} C_VEL
LIN {X 0,Y 379.979,Z 702.936,A -85,B 0,C 180,E1 -10278.566,E2 -10278.566} C_VEL
LIN {X 0,Y 381.705,Z 690.726,A -85,B 0,C 180,E1 -10280.87,E2 -10280.87} C_VEL
LIN {X 0,Y 383.685,Z 677.062,A -85,B 0,C 180,E1 -10283.011,E2 -10283.011} C_VEL
LIN {X 0,Y 385.869,Z 661.873,A -85,B 0,C 180,E1 -10284.985,E2 -10284.985} C_VEL
LIN {X 0,Y 388.085,Z 645.73,A -85,B 0,C 180,E1 -10286.717,E2 -10286.717} C_VEL
LIN {X 0,Y 390.283,Z 628.511,A -85,B 0,C 180,E1 -10288.231,E2 -10288.231} C_VEL
LIN {X 0,Y 392.391,Z 609.893,A -85,B 0,C 180,E1 -10289.545,E2 -10289.545} C_VEL
LIN {X 0,Y 394.273,Z 590.391,A -85,B 0,C 180,E1 -10290.609,E2 -10290.609} C_VEL
LIN {X 0,Y 395.803,Z 570.164,A -85,B 0,C 180,E1 -10291.412,E2 -10291.412} C_VEL
LIN {X 0,Y 396.936,Z 548.319,A -85,B 0,C 180,E1 -10291.985,E2 -10291.985} C_VEL
LIN {X 0,Y 404.242,Z 376.052,A -85,B 0,C 180,E1 -10295.8,E2 -10295.8} C_VEL
LIN {X 0,Y 399.757,Z 345.342,A -85,B 0,C 180,E1 -10297.071,E2 -10297.071} C_VEL
LIN {X 0,Y 396.829,Z 339.435,A -85,B 0,C 180,E1 -10297.572,E2 -10297.572} C_VEL
LIN {X 0,Y 389.659,Z 319.65,A -85,B 0,C 180,E1 -10300.801,E2 -10300.801} C_VEL
LIN {X 0,Y 382.005,Z 300.218,A -85,B 0,C 180,E1 -10304.285,E2 -10304.285} C_VEL
LIN {X 0,Y 377.705,Z 289.65,A -85,B 0,C 180,E1 -10306.365,E2 -10306.365} C_VEL
LIN {X 0,Y 377.684,Z 289.439,A -85,B 0,C 180,E1 -10310.389,E2 -10310.389} C_VEL
LIN {X 0,Y 377.682,Z 289.441,A -85,B 0,C 180,E1 -10314.378,E2 -10314.378} C_VEL
LIN {X 0,Y 377.683,Z 289.439,A -85,B 0,C 180,E1 -10318.48,E2 -10318.48} C_VEL
LIN {X 0,Y 377.673,Z 289.44,A -85,B 0,C 180,E1 -10322.569,E2 -10322.569} C_VEL
LIN {X 0,Y 377.665,Z 289.439,A -85,B 0,C 180,E1 -10326.6,E2 -10326.6} C_VEL
LIN {X 0,Y 377.702,Z 289.655,A -85,B 0,C 180,E1 -10329.647,E2 -10329.647} C_VEL
LIN {X 0,Y 385.933,Z 309.834,A -85,B 0,C 180,E1 -10332.743,E2 -10332.743} C_VEL
LIN {X 0,Y 392.695,Z 328.668,A -85,B 0,C 180,E1 -10335.363,E2 -10335.363} C_VEL
LIN {X 0,Y 395.707,Z 338.188,A -85,B 0,C 180,E1 -10336.61,E2 -10336.61} C_VEL
LIN {X 0,Y 393.42,Z 376.867,A -85,B 0,C 180,E1 -10340.245,E2 -10340.245} C_VEL
LIN {X 0,Y 392.128,Z 383.541,A -85,B 0,C 180,E1 -10340.792,E2 -10340.792} C_VEL
LIN {X 0,Y 385.455,Z 401.884,A -85,B 0,C 180,E1 -10342.039,E2 -10342.039} C_VEL
LIN {X 0,Y 384.433,Z 407.611,A -85,B 0,C 180,E1 -10342.525,E2 -10342.525} C_VEL
LIN {X 0,Y 381.606,Z 451.549,A -85,B 0,C 180,E1 -10346.694,E2 -10346.694} C_VEL
LIN {X 0,Y 379.974,Z 480.131,A -85,B 0,C 180,E1 -10349.371,E2 -10349.371} C_VEL
LIN {X 0,Y 381.841,Z 498.458,A -85,B 0,C 180,E1 -10349.884,E2 -10349.884} C_VEL
LIN {X 0,Y 379.17,Z 623.534,A -85,B 0,C 180,E1 -10352.317,E2 -10352.317} C_VEL
LIN {X 0,Y 378.494,Z 639.636,A -85,B 0,C 180,E1 -10352.909,E2 -10352.909} C_VEL
LIN {X 0,Y 377.466,Z 655.734,A -85,B 0,C 180,E1 -10353.795,E2 -10353.795} C_VEL
LIN {X 0,Y 376.243,Z 670.094,A -85,B 0,C 180,E1 -10354.877,E2 -10354.877} C_VEL
LIN {X 0,Y 374.792,Z 684.434,A -85,B 0,C 180,E1 -10356.278,E2 -10356.278} C_VEL
LIN {X 0,Y 373.359,Z 697.059,A -85,B 0,C 180,E1 -10357.848,E2 -10357.848} C_VEL
LIN {X 0,Y 371.897,Z 709.206,A -85,B 0,C 180,E1 -10359.75,E2 -10359.75} C_VEL
LIN {X 0,Y 370.678,Z 719.166,A -85,B 0,C 180,E1 -10361.718,E2 -10361.718} C_VEL
LIN {X 0,Y 369.647,Z 727.998,A -85,B 0,C 180,E1 -10363.928,E2 -10363.928} C_VEL
LIN {X 0,Y 368.914,Z 734.996,A -85,B 0,C 180,E1 -10366.208,E2 -10366.208} C_VEL
LIN {X 0,Y 368.428,Z 740.585,A -85,B 0,C 180,E1 -10368.711,E2 -10368.711} C_VEL
LIN {X 0,Y 368.192,Z 744.202,A -85,B 0,C 180,E1 -10371.17,E2 -10371.17} C_VEL
LIN {X 0,Y 368.104,Z 746.127,A -85,B 0,C 180,E1 -10373.739,E2 -10373.739} C_VEL
LIN {X 0,Y 368.109,Z 746.272,A -85,B 0,C 180,E1 -10376.277,E2 -10376.277} C_VEL
LIN {X 0,Y 368.211,Z 744.521,A -85,B 0,C 180,E1 -10378.902,E2 -10378.902} C_VEL
LIN {X 0,Y 368.472,Z 741.087,A -85,B 0,C 180,E1 -10381.397,E2 -10381.397} C_VEL
LIN {X 0,Y 368.99,Z 735.613,A -85,B 0,C 180,E1 -10383.929,E2 -10383.929} C_VEL
LIN {X 0,Y 369.729,Z 729.147,A -85,B 0,C 180,E1 -10386.121,E2 -10386.121} C_VEL
LIN {X 0,Y 370.786,Z 720.614,A -85,B 0,C 180,E1 -10388.329,E2 -10388.329} C_VEL
LIN {X 0,Y 372.085,Z 710.69,A -85,B 0,C 180,E1 -10390.359,E2 -10390.359} C_VEL
LIN {X 0,Y 373.545,Z 699.243,A -85,B 0,C 180,E1 -10392.207,E2 -10392.207} C_VEL
LIN {X 0,Y 375.103,Z 686.352,A -85,B 0,C 180,E1 -10393.869,E2 -10393.869} C_VEL
LIN {X 0,Y 376.6,Z 672.251,A -85,B 0,C 180,E1 -10395.285,E2 -10395.285} C_VEL
LIN {X 0,Y 377.971,Z 657.195,A -85,B 0,C 180,E1 -10396.451,E2 -10396.451} C_VEL
LIN {X 0,Y 379.05,Z 640.978,A -85,B 0,C 180,E1 -10397.359,E2 -10397.359} C_VEL
LIN {X 0,Y 379.755,Z 624.876,A -85,B 0,C 180,E1 -10397.967,E2 -10397.967} C_VEL
LIN {X 0,Y 381.195,Z 558.96,A -85,B 0,C 180,E1 -10399.284,E2 -10399.284} C_VEL
LIN {X 0,Y 382.467,Z 495.618,A -85,B 0,C 180,E1 -10400.524,E2 -10400.524} C_VEL
LIN {X 0,Y 380.711,Z 480.143,A -85,B 0,C 180,E1 -10401.018,E2 -10401.018} C_VEL
LIN {X 0,Y 383.378,Z 436.859,A -85,B 0,C 180,E1 -10405.077,E2 -10405.077} C_VEL
LIN {X 0,Y 385.959,Z 395.249,A -85,B 0,C 180,E1 -10408.967,E2 -10408.967} C_VEL
LIN {X 0,Y 388.328,Z 354.742,A -85,B 0,C 180,E1 -10412.721,E2 -10412.721} C_VEL
LIN {X 0,Y 389.068,Z 340.012,A -85,B 0,C 180,E1 -10414.094,E2 -10414.094} C_VEL
LIN {X 0,Y 383.738,Z 323.637,A -85,B 0,C 180,E1 -10416.342,E2 -10416.342} C_VEL
LIN {X 0,Y 377.887,Z 308.744,A -85,B 0,C 180,E1 -10418.583,E2 -10418.583} C_VEL
LIN {X 0,Y 371.317,Z 294.299,A -85,B 0,C 180,E1 -10420.984,E2 -10420.984} C_VEL
LIN {X 0,Y 369.768,Z 290.793,A -85,B 0,C 180,E1 -10421.635,E2 -10421.635} C_VEL
LIN {X 0,Y 369.741,Z 290.423,A -85,B 0,C 180,E1 -10422.369,E2 -10422.369} C_VEL
LIN {X 0,Y 369.751,Z 290.433,A -85,B 0,C 180,E1 -10426.552,E2 -10426.552} C_VEL
LIN {X 0,Y 369.746,Z 290.428,A -85,B 0,C 180,E1 -10430.745,E2 -10430.745} C_VEL
LIN {X 0,Y 369.746,Z 290.43,A -85,B 0,C 180,E1 -10434.724,E2 -10434.724} C_VEL
LIN {X 0,Y 369.746,Z 290.425,A -85,B 0,C 180,E1 -10438.915,E2 -10438.915} C_VEL
LIN {X 0,Y 369.741,Z 290.427,A -85,B 0,C 180,E1 -10442.945,E2 -10442.945} C_VEL
LIN {X 0,Y 369.746,Z 290.423,A -85,B 0,C 180,E1 -10447.073,E2 -10447.073} C_VEL
LIN {X 0,Y 369.735,Z 290.429,A -85,B 0,C 180,E1 -10451.227,E2 -10451.227} C_VEL
LIN {X 0,Y 369.742,Z 290.423,A -85,B 0,C 180,E1 -10455.207,E2 -10455.207} C_VEL
LIN {X 0,Y 369.737,Z 290.424,A -85,B 0,C 180,E1 -10459.311,E2 -10459.311} C_VEL
LIN {X 0,Y 369.735,Z 290.429,A -85,B 0,C 180,E1 -10463.423,E2 -10463.423} C_VEL
LIN {X 0,Y 369.731,Z 290.426,A -85,B 0,C 180,E1 -10467.544,E2 -10467.544} C_VEL
LIN {X 0,Y 369.733,Z 290.427,A -85,B 0,C 180,E1 -10471.592,E2 -10471.592} C_VEL
LIN {X 0,Y 369.727,Z 290.428,A -85,B 0,C 180,E1 -10475.741,E2 -10475.741} C_VEL
LIN {X 0,Y 369.775,Z 290.691,A -85,B 0,C 180,E1 -10479.587,E2 -10479.587} C_VEL
LIN {X 0,Y 372.529,Z 297.351,A -85,B 0,C 180,E1 -10480.911,E2 -10480.911} C_VEL
LIN {X 0,Y 380.514,Z 315.687,A -85,B 0,C 180,E1 -10484.238,E2 -10484.238} C_VEL
LIN {X 0,Y 382.502,Z 320.216,A -85,B 0,C 180,E1 -10484.945,E2 -10484.945} C_VEL
LIN {X 0,Y 398.543,Z 348.214,A -85,B 0,C 180,E1 -10487.552,E2 -10487.552} C_VEL
LIN {X 0,Y 403.094,Z 356.879,A -85,B 0,C 180,E1 -10488.271,E2 -10488.271} C_VEL
LIN {X 0,Y 394.051,Z 557.218,A -85,B 0,C 180,E1 -10492.65,E2 -10492.65} C_VEL
LIN {X 0,Y 392.751,Z 582.341,A -85,B 0,C 180,E1 -10493.276,E2 -10493.276} C_VEL
LIN {X 0,Y 390.974,Z 603.771,A -85,B 0,C 180,E1 -10494.07,E2 -10494.07} C_VEL
LIN {X 0,Y 388.828,Z 624.372,A -85,B 0,C 180,E1 -10495.114,E2 -10495.114} C_VEL
LIN {X 0,Y 386.349,Z 644.626,A -85,B 0,C 180,E1 -10496.441,E2 -10496.441} C_VEL
LIN {X 0,Y 383.787,Z 663.16,A -85,B 0,C 180,E1 -10497.95,E2 -10497.95} C_VEL
LIN {X 0,Y 381.235,Z 680.303,A -85,B 0,C 180,E1 -10499.639,E2 -10499.639} C_VEL
LIN {X 0,Y 378.598,Z 697.08,A -85,B 0,C 180,E1 -10501.619,E2 -10501.619} C_VEL
LIN {X 0,Y 376.01,Z 713.155,A -85,B 0,C 180,E1 -10503.893,E2 -10503.893} C_VEL
LIN {X 0,Y 373.725,Z 727.589,A -85,B 0,C 180,E1 -10506.342,E2 -10506.342} C_VEL
LIN {X 0,Y 371.736,Z 740.831,A -85,B 0,C 180,E1 -10509.041,E2 -10509.041} C_VEL
LIN {X 0,Y 370.249,Z 751.822,A -85,B 0,C 180,E1 -10511.746,E2 -10511.746} C_VEL
LIN {X 0,Y 369.161,Z 761.382,A -85,B 0,C 180,E1 -10514.61,E2 -10514.61} C_VEL
LIN {X 0,Y 368.458,Z 769.429,A -85,B 0,C 180,E1 -10517.623,E2 -10517.623} C_VEL
LIN {X 0,Y 368.119,Z 775.579,A -85,B 0,C 180,E1 -10520.623,E2 -10520.623} C_VEL
LIN {X 0,Y 368.022,Z 779.808,A -85,B 0,C 180,E1 -10523.45,E2 -10523.45} C_VEL
LIN {X 0,Y 368.02,Z 782.534,A -85,B 0,C 180,E1 -10526.419,E2 -10526.419} C_VEL
LIN {X 0,Y 368.043,Z 783.64,A -85,B 0,C 180,E1 -10529.379,E2 -10529.379} C_VEL
LIN {X 0,Y 368.035,Z 783.149,A -85,B 0,C 180,E1 -10532.337,E2 -10532.337} C_VEL
LIN {X 0,Y 368.011,Z 781.189,A -85,B 0,C 180,E1 -10535.146,E2 -10535.146} C_VEL
LIN {X 0,Y 368.069,Z 777.445,A -85,B 0,C 180,E1 -10538.122,E2 -10538.122} C_VEL
LIN {X 0,Y 368.282,Z 771.99,A -85,B 0,C 180,E1 -10541.115,E2 -10541.115} C_VEL
LIN {X 0,Y 368.805,Z 764.701,A -85,B 0,C 180,E1 -10544.124,E2 -10544.124} C_VEL
LIN {X 0,Y 369.691,Z 755.961,A -85,B 0,C 180,E1 -10546.985,E2 -10546.985} C_VEL
LIN {X 0,Y 371.059,Z 745.069,A -85,B 0,C 180,E1 -10549.879,E2 -10549.879} C_VEL
LIN {X 0,Y 372.804,Z 732.852,A -85,B 0,C 180,E1 -10552.554,E2 -10552.554} C_VEL
LIN {X 0,Y 374.959,Z 718.978,A -85,B 0,C 180,E1 -10555.088,E2 -10555.088} C_VEL
LIN {X 0,Y 377.339,Z 704.103,A -85,B 0,C 180,E1 -10557.371,E2 -10557.371} C_VEL
LIN {X 0,Y 379.992,Z 687.829,A -85,B 0,C 180,E1 -10559.477,E2 -10559.477} C_VEL
LIN {X 0,Y 382.806,Z 670.038,A -85,B 0,C 180,E1 -10561.406,E2 -10561.406} C_VEL
LIN {X 0,Y 385.753,Z 650.514,A -85,B 0,C 180,E1 -10563.156,E2 -10563.156} C_VEL
LIN {X 0,Y 388.648,Z 629.964,A -85,B 0,C 180,E1 -10564.651,E2 -10564.651} C_VEL
LIN {X 0,Y 391.397,Z 608.329,A -85,B 0,C 180,E1 -10565.904,E2 -10565.904} C_VEL
LIN {X 0,Y 393.844,Z 586.698,A -85,B 0,C 180,E1 -10566.855,E2 -10566.855} C_VEL
LIN {X 0,Y 395.974,Z 562.993,A -85,B 0,C 180,E1 -10567.617,E2 -10567.617} C_VEL
LIN {X 0,Y 400.952,Z 503.872,A -85,B 0,C 180,E1 -10569.286,E2 -10569.286} C_VEL
LIN {X 0,Y 407.588,Z 446.434,A -85,B 0,C 180,E1 -10571.053,E2 -10571.053} C_VEL
LIN {X 0,Y 416.346,Z 388.579,A -85,B 0,C 180,E1 -10572.921,E2 -10572.921} C_VEL
LIN {X 0,Y 420.44,Z 365.452,A -85,B 0,C 180,E1 -10573.702,E2 -10573.702} C_VEL
LIN {X 0,Y 419.53,Z 363.016,A -85,B 0,C 180,E1 -10574.554,E2 -10574.554} C_VEL
LIN {X 0,Y 418.737,Z 360.955,A -85,B 0,C 180,E1 -10575.795,E2 -10575.795} C_VEL
LIN {X 0,Y 418.331,Z 361.229,A -85,B 0,C 180,E1 -10576.689,E2 -10576.689} C_VEL
LIN {X 0,Y 418.348,Z 363.199,A -85,B 0,C 180,E1 -10578.087,E2 -10578.087} C_VEL
LIN {X 0,Y 419.16,Z 367.683,A -85,B 0,C 180,E1 -10579.601,E2 -10579.601} C_VEL
LIN {X 0,Y 419.383,Z 369.481,A -85,B 0,C 180,E1 -10579.965,E2 -10579.965} C_VEL
LIN {X 0,Y 418.006,Z 383.821,A -85,B 0,C 180,E1 -10581.007,E2 -10581.007} C_VEL
LIN {X 0,Y 406.652,Z 454.241,A -85,B 0,C 180,E1 -10583.338,E2 -10583.338} C_VEL
LIN {X 0,Y 398.55,Z 518.695,A -85,B 0,C 180,E1 -10585.45,E2 -10585.45} C_VEL
LIN {X 0,Y 393.19,Z 572.044,A -85,B 0,C 180,E1 -10587.172,E2 -10587.172} C_VEL
LIN {X 0,Y 390.813,Z 592.528,A -85,B 0,C 180,E1 -10588.109,E2 -10588.109} C_VEL
LIN {X 0,Y 388.137,Z 612.992,A -85,B 0,C 180,E1 -10589.333,E2 -10589.333} C_VEL
LIN {X 0,Y 385.32,Z 632.248,A -85,B 0,C 180,E1 -10590.802,E2 -10590.802} C_VEL
LIN {X 0,Y 382.563,Z 649.759,A -85,B 0,C 180,E1 -10592.445,E2 -10592.445} C_VEL
LIN {X 0,Y 379.805,Z 666.333,A -85,B 0,C 180,E1 -10594.339,E2 -10594.339} C_VEL
LIN {X 0,Y 377.138,Z 681.804,A -85,B 0,C 180,E1 -10596.485,E2 -10596.485} C_VEL
LIN {X 0,Y 374.817,Z 695.181,A -85,B 0,C 180,E1 -10598.729,E2 -10598.729} C_VEL
LIN {X 0,Y 372.735,Z 707.431,A -85,B 0,C 180,E1 -10601.223,E2 -10601.223} C_VEL
LIN {X 0,Y 371.118,Z 717.485,A -85,B 0,C 180,E1 -10603.729,E2 -10603.729} C_VEL
LIN {X 0,Y 369.861,Z 726.123,A -85,B 0,C 180,E1 -10606.398,E2 -10606.398} C_VEL
LIN {X 0,Y 368.975,Z 733.258,A -85,B 0,C 180,E1 -10609.224,E2 -10609.224} C_VEL
LIN {X 0,Y 368.446,Z 738.52,A -85,B 0,C 180,E1 -10612.045,E2 -10612.045} C_VEL
LIN {X 0,Y 368.187,Z 742.055,A -85,B 0,C 180,E1 -10614.859,E2 -10614.859} C_VEL
LIN {X 0,Y 368.078,Z 743.947,A -85,B 0,C 180,E1 -10617.665,E2 -10617.665} C_VEL
LIN {X 0,Y 368.051,Z 744.24,A -85,B 0,C 180,E1 -10620.468,E2 -10620.468} C_VEL
LIN {X 0,Y 368.066,Z 742.931,A -85,B 0,C 180,E1 -10623.271,E2 -10623.271} C_VEL
LIN {X 0,Y 368.166,Z 740.004,A -85,B 0,C 180,E1 -10626.081,E2 -10626.081} C_VEL
LIN {X 0,Y 368.438,Z 735.283,A -85,B 0,C 180,E1 -10628.948,E2 -10628.948} C_VEL
LIN {X 0,Y 368.976,Z 728.947,A -85,B 0,C 180,E1 -10631.727,E2 -10631.727} C_VEL
LIN {X 0,Y 369.827,Z 721.055,A -85,B 0,C 180,E1 -10634.403,E2 -10634.403} C_VEL
LIN {X 0,Y 371.003,Z 711.81,A -85,B 0,C 180,E1 -10636.922,E2 -10636.922} C_VEL
LIN {X 0,Y 372.593,Z 700.493,A -85,B 0,C 180,E1 -10639.437,E2 -10639.437} C_VEL
LIN {X 0,Y 374.5,Z 687.664,A -85,B 0,C 180,E1 -10641.785,E2 -10641.785} C_VEL
LIN {X 0,Y 376.673,Z 673.272,A -85,B 0,C 180,E1 -10643.963,E2 -10643.963} C_VEL
LIN {X 0,Y 378.915,Z 658.124,A -85,B 0,C 180,E1 -10645.865,E2 -10645.865} C_VEL
LIN {X 0,Y 381.192,Z 641.872,A -85,B 0,C 180,E1 -10647.553,E2 -10647.553} C_VEL
LIN {X 0,Y 383.414,Z 624.653,A -85,B 0,C 180,E1 -10649.016,E2 -10649.016} C_VEL
LIN {X 0,Y 385.514,Z 606.259,A -85,B 0,C 180,E1 -10650.268,E2 -10650.268} C_VEL
LIN {X 0,Y 387.38,Z 586.654,A -85,B 0,C 180,E1 -10651.297,E2 -10651.297} C_VEL
LIN {X 0,Y 388.941,Z 566.164,A -85,B 0,C 180,E1 -10652.069,E2 -10652.069} C_VEL
LIN {X 0,Y 390.345,Z 536.46,A -85,B 0,C 180,E1 -10652.796,E2 -10652.796} C_VEL
LIN {X 0,Y 397.577,Z 377.275,A -85,B 0,C 180,E1 -10656.419,E2 -10656.419} C_VEL
LIN {X 0,Y 393.441,Z 348.721,A -85,B 0,C 180,E1 -10657.631,E2 -10657.631} C_VEL
LIN {X 0,Y 388.564,Z 339.103,A -85,B 0,C 180,E1 -10658.471,E2 -10658.471} C_VEL
LIN {X 0,Y 381.373,Z 319.703,A -85,B 0,C 180,E1 -10661.754,E2 -10661.754} C_VEL
LIN {X 0,Y 374.161,Z 301.415,A -85,B 0,C 180,E1 -10665.13,E2 -10665.13} C_VEL
LIN {X 0,Y 369.778,Z 290.655,A -85,B 0,C 180,E1 -10667.316,E2 -10667.316} C_VEL
LIN {X 0,Y 369.749,Z 290.429,A -85,B 0,C 180,E1 -10671.399,E2 -10671.399} C_VEL
LIN {X 0,Y 369.743,Z 290.426,A -85,B 0,C 180,E1 -10675.584,E2 -10675.584} C_VEL
LIN {X 0,Y 369.747,Z 290.411,A -85,B 0,C 180,E1 -10679.622,E2 -10679.622} C_VEL
LIN {X 0,Y 369.739,Z 290.421,A -85,B 0,C 180,E1 -10683.672,E2 -10683.672} C_VEL
LIN {X 0,Y 369.744,Z 290.418,A -85,B 0,C 180,E1 -10687.752,E2 -10687.752} C_VEL
LIN {X 0,Y 369.75,Z 290.681,A -85,B 0,C 180,E1 -10688.795,E2 -10688.795} C_VEL
LIN {X 0,Y 378.347,Z 311.374,A -85,B 0,C 180,E1 -10692.061,E2 -10692.061} C_VEL
LIN {X 0,Y 385.096,Z 329.918,A -85,B 0,C 180,E1 -10694.719,E2 -10694.719} C_VEL
LIN {X 0,Y 388.637,Z 341.241,A -85,B 0,C 180,E1 -10696.231,E2 -10696.231} C_VEL
LIN {X 0,Y 386.021,Z 382.579,A -85,B 0,C 180,E1 -10700.155,E2 -10700.155} C_VEL
LIN {X 0,Y 384.433,Z 407.611,A -85,B 0,C 180,E1 -10702.525,E2 -10702.525} C_VEL
LIN {X 0,Y 383.132,Z 414.289,A -85,B 0,C 180,E1 -10703.083,E2 -10703.083} C_VEL
LIN {X 0,Y 376.341,Z 432.592,A -85,B 0,C 180,E1 -10704.355,E2 -10704.355} C_VEL
LIN {X 0,Y 375.3,Z 438.327,A -85,B 0,C 180,E1 -10704.849,E2 -10704.849} C_VEL
LIN {X 0,Y 372.631,Z 480.345,A -85,B 0,C 180,E1 -10708.85,E2 -10708.85} C_VEL
LIN {X 0,Y 374.555,Z 499.287,A -85,B 0,C 180,E1 -10709.391,E2 -10709.391} C_VEL
LIN {X 0,Y 371.744,Z 623.954,A -85,B 0,C 180,E1 -10711.867,E2 -10711.867} C_VEL
LIN {X 0,Y 371.04,Z 640.012,A -85,B 0,C 180,E1 -10712.469,E2 -10712.469} C_VEL
LIN {X 0,Y 369.982,Z 655.877,A -85,B 0,C 180,E1 -10713.357,E2 -10713.357} C_VEL
LIN {X 0,Y 368.737,Z 669.994,A -85,B 0,C 180,E1 -10714.43,E2 -10714.43} C_VEL
LIN {X 0,Y 367.225,Z 684.313,A -85,B 0,C 180,E1 -10715.846,E2 -10715.846} C_VEL
LIN {X 0,Y 365.703,Z 697.159,A -85,B 0,C 180,E1 -10717.46,E2 -10717.46} C_VEL
LIN {X 0,Y 364.22,Z 708.895,A -85,B 0,C 180,E1 -10719.319,E2 -10719.319} C_VEL
LIN {X 0,Y 362.949,Z 718.813,A -85,B 0,C 180,E1 -10721.277,E2 -10721.277} C_VEL
LIN {X 0,Y 361.809,Z 727.957,A -85,B 0,C 180,E1 -10723.584,E2 -10723.584} C_VEL
LIN {X 0,Y 361.014,Z 735.082,A -85,B 0,C 180,E1 -10725.912,E2 -10725.912} C_VEL
LIN {X 0,Y 360.481,Z 740.708,A -85,B 0,C 180,E1 -10728.448,E2 -10728.448} C_VEL
LIN {X 0,Y 360.22,Z 744.468,A -85,B 0,C 180,E1 -10730.979,E2 -10730.979} C_VEL
LIN {X 0,Y 360.115,Z 746.468,A -85,B 0,C 180,E1 -10733.615,E2 -10733.615} C_VEL
LIN {X 0,Y 360.118,Z 746.707,A -85,B 0,C 180,E1 -10736.195,E2 -10736.195} C_VEL
LIN {X 0,Y 360.212,Z 745.207,A -85,B 0,C 180,E1 -10738.699,E2 -10738.699} C_VEL
LIN {X 0,Y 360.482,Z 741.88,A -85,B 0,C 180,E1 -10741.317,E2 -10741.317} C_VEL
LIN {X 0,Y 360.99,Z 736.788,A -85,B 0,C 180,E1 -10743.827,E2 -10743.827} C_VEL
LIN {X 0,Y 361.814,Z 729.961,A -85,B 0,C 180,E1 -10746.252,E2 -10746.252} C_VEL
LIN {X 0,Y 362.929,Z 721.526,A -85,B 0,C 180,E1 -10748.517,E2 -10748.517} C_VEL
LIN {X 0,Y 364.342,Z 711.321,A -85,B 0,C 180,E1 -10750.663,E2 -10750.663} C_VEL
LIN {X 0,Y 365.805,Z 700.533,A -85,B 0,C 180,E1 -10752.461,E2 -10752.461} C_VEL
LIN {X 0,Y 367.422,Z 687.824,A -85,B 0,C 180,E1 -10754.156,E2 -10754.156} C_VEL
LIN {X 0,Y 368.904,Z 674.932,A -85,B 0,C 180,E1 -10755.523,E2 -10755.523} C_VEL
LIN {X 0,Y 370.302,Z 660.652,A -85,B 0,C 180,E1 -10756.698,E2 -10756.698} C_VEL
LIN {X 0,Y 371.494,Z 645.139,A -85,B 0,C 180,E1 -10757.659,E2 -10757.659} C_VEL
LIN {X 0,Y 372.331,Z 628.571,A -85,B 0,C 180,E1 -10758.355,E2 -10758.355} C_VEL
LIN {X 0,Y 372.829,Z 609.797,A -85,B 0,C 180,E1 -10758.811,E2 -10758.811} C_VEL
LIN {X 0,Y 375.331,Z 496.579,A -85,B 0,C 180,E1 -10761.057,E2 -10761.057} C_VEL
LIN {X 0,Y 373.529,Z 480.228,A -85,B 0,C 180,E1 -10761.609,E2 -10761.609} C_VEL
LIN {X 0,Y 376.355,Z 437.011,A -85,B 0,C 180,E1 -10765.709,E2 -10765.709} C_VEL
LIN {X 0,Y 379.094,Z 395.27,A -85,B 0,C 180,E1 -10769.654,E2 -10769.654} C_VEL
LIN {X 0,Y 381.738,Z 352.371,A -85,B 0,C 180,E1 -10773.671,E2 -10773.671} C_VEL
LIN {X 0,Y 382.179,Z 342.798,A -85,B 0,C 180,E1 -10774.592,E2 -10774.592} C_VEL
LIN {X 0,Y 376.531,Z 325.559,A -85,B 0,C 180,E1 -10777.023,E2 -10777.023} C_VEL
LIN {X 0,Y 370.306,Z 310.03,A -85,B 0,C 180,E1 -10779.45,E2 -10779.45} C_VEL
LIN {X 0,Y 364.847,Z 298.49,A -85,B 0,C 180,E1 -10781.464,E2 -10781.464} C_VEL
LIN {X 0,Y 361.863,Z 291.816,A -85,B 0,C 180,E1 -10782.72,E2 -10782.72} C_VEL
LIN {X 0,Y 361.776,Z 291.421,A -85,B 0,C 180,E1 -10783.295,E2 -10783.295} C_VEL
LIN {X 0,Y 361.777,Z 291.421,A -85,B 0,C 180,E1 -10787.388,E2 -10787.388} C_VEL
LIN {X 0,Y 361.775,Z 291.418,A -85,B 0,C 180,E1 -10791.576,E2 -10791.576} C_VEL
LIN {X 0,Y 361.776,Z 291.417,A -85,B 0,C 180,E1 -10795.72,E2 -10795.72} C_VEL
LIN {X 0,Y 361.777,Z 291.421,A -85,B 0,C 180,E1 -10799.841,E2 -10799.841} C_VEL
LIN {X 0,Y 361.777,Z 291.414,A -85,B 0,C 180,E1 -10803.961,E2 -10803.961} C_VEL
LIN {X 0,Y 361.78,Z 291.42,A -85,B 0,C 180,E1 -10808.102,E2 -10808.102} C_VEL
LIN {X 0,Y 361.786,Z 291.414,A -85,B 0,C 180,E1 -10812.286,E2 -10812.286} C_VEL
LIN {X 0,Y 361.79,Z 291.413,A -85,B 0,C 180,E1 -10816.373,E2 -10816.373} C_VEL
LIN {X 0,Y 361.799,Z 291.42,A -85,B 0,C 180,E1 -10820.546,E2 -10820.546} C_VEL
LIN {X 0,Y 361.801,Z 291.414,A -85,B 0,C 180,E1 -10824.664,E2 -10824.664} C_VEL
LIN {X 0,Y 361.818,Z 291.415,A -85,B 0,C 180,E1 -10828.92,E2 -10828.92} C_VEL
LIN {X 0,Y 361.809,Z 291.418,A -85,B 0,C 180,E1 -10833.144,E2 -10833.144} C_VEL
LIN {X 0,Y 361.808,Z 291.417,A -85,B 0,C 180,E1 -10837.265,E2 -10837.265} C_VEL
LIN {X 0,Y 361.853,Z 291.791,A -85,B 0,C 180,E1 -10838.601,E2 -10838.601} C_VEL
LIN {X 0,Y 370.051,Z 310.673,A -85,B 0,C 180,E1 -10842.282,E2 -10842.282} C_VEL
LIN {X 0,Y 374.269,Z 320.363,A -85,B 0,C 180,E1 -10843.967,E2 -10843.967} C_VEL
LIN {X 0,Y 391.264,Z 349.93,A -85,B 0,C 180,E1 -10846.824,E2 -10846.824} C_VEL
LIN {X 0,Y 396.467,Z 359.906,A -85,B 0,C 180,E1 -10847.662,E2 -10847.662} C_VEL
LIN {X 0,Y 387.034,Z 557.79,A -85,B 0,C 180,E1 -10852.091,E2 -10852.091} C_VEL
LIN {X 0,Y 385.672,Z 582.621,A -85,B 0,C 180,E1 -10852.729,E2 -10852.729} C_VEL
LIN {X 0,Y 383.819,Z 604.013,A -85,B 0,C 180,E1 -10853.542,E2 -10853.542} C_VEL
LIN {X 0,Y 381.572,Z 624.706,A -85,B 0,C 180,E1 -10854.615,E2 -10854.615} C_VEL
LIN {X 0,Y 378.957,Z 645.216,A -85,B 0,C 180,E1 -10855.992,E2 -10855.992} C_VEL
LIN {X 0,Y 376.163,Z 664.59,A -85,B 0,C 180,E1 -10857.618,E2 -10857.618} C_VEL
LIN {X 0,Y 373.295,Z 682.905,A -85,B 0,C 180,E1 -10859.5,E2 -10859.5} C_VEL
LIN {X 0,Y 370.468,Z 700.128,A -85,B 0,C 180,E1 -10861.643,E2 -10861.643} C_VEL
LIN {X 0,Y 367.863,Z 715.674,A -85,B 0,C 180,E1 -10863.965,E2 -10863.965} C_VEL
LIN {X 0,Y 365.568,Z 729.69,A -85,B 0,C 180,E1 -10866.466,E2 -10866.466} C_VEL
LIN {X 0,Y 363.692,Z 741.895,A -85,B 0,C 180,E1 -10869.062,E2 -10869.062} C_VEL
LIN {X 0,Y 362.195,Z 752.719,A -85,B 0,C 180,E1 -10871.826,E2 -10871.826} C_VEL
LIN {X 0,Y 361.109,Z 762.048,A -85,B 0,C 180,E1 -10874.751,E2 -10874.751} C_VEL
LIN {X 0,Y 360.45,Z 769.492,A -85,B 0,C 180,E1 -10877.669,E2 -10877.669} C_VEL
LIN {X 0,Y 360.116,Z 775.518,A -85,B 0,C 180,E1 -10880.735,E2 -10880.735} C_VEL
LIN {X 0,Y 360.029,Z 779.619,A -85,B 0,C 180,E1 -10883.624,E2 -10883.624} C_VEL
LIN {X 0,Y 360.031,Z 782.152,A -85,B 0,C 180,E1 -10886.499,E2 -10886.499} C_VEL
LIN {X 0,Y 360.056,Z 783.184,A -85,B 0,C 180,E1 -10889.365,E2 -10889.365} C_VEL
LIN {X 0,Y 360.046,Z 782.801,A -85,B 0,C 180,E1 -10892.23,E2 -10892.23} C_VEL
LIN {X 0,Y 360.019,Z 780.891,A -85,B 0,C 180,E1 -10895.1,E2 -10895.1} C_VEL
LIN {X 0,Y 360.071,Z 777.255,A -85,B 0,C 180,E1 -10898.143,E2 -10898.143} C_VEL
LIN {X 0,Y 360.29,Z 771.904,A -85,B 0,C 180,E1 -10901.203,E2 -10901.203} C_VEL
LIN {X 0,Y 360.802,Z 765.169,A -85,B 0,C 180,E1 -10904.116,E2 -10904.116} C_VEL
LIN {X 0,Y 361.715,Z 756.614,A -85,B 0,C 180,E1 -10907.04,E2 -10907.04} C_VEL
LIN {X 0,Y 363.113,Z 746.047,A -85,B 0,C 180,E1 -10909.966,E2 -10909.966} C_VEL
LIN {X 0,Y 364.945,Z 733.976,A -85,B 0,C 180,E1 -10912.726,E2 -10912.726} C_VEL
LIN {X 0,Y 367.19,Z 720.436,A -85,B 0,C 180,E1 -10915.311,E2 -10915.311} C_VEL
LIN {X 0,Y 369.866,Z 704.884,A -85,B 0,C 180,E1 -10917.797,E2 -10917.797} C_VEL
LIN {X 0,Y 372.777,Z 688.278,A -85,B 0,C 180,E1 -10920.017,E2 -10920.017} C_VEL
LIN {X 0,Y 375.897,Z 670.021,A -85,B 0,C 180,E1 -10922.051,E2 -10922.051} C_VEL
LIN {X 0,Y 379.18,Z 649.853,A -85,B 0,C 180,E1 -10923.899,E2 -10923.899} C_VEL
LIN {X 0,Y 382.324,Z 629.272,A -85,B 0,C 180,E1 -10925.427,E2 -10925.427} C_VEL
LIN {X 0,Y 385.372,Z 607.362,A -85,B 0,C 180,E1 -10926.722,E2 -10926.722} C_VEL
LIN {X 0,Y 388.095,Z 585.513,A -85,B 0,C 180,E1 -10927.703,E2 -10927.703} C_VEL
LIN {X 0,Y 390.531,Z 561.018,A -85,B 0,C 180,E1 -10928.509,E2 -10928.509} C_VEL
LIN {X 0,Y 396.15,Z 504.027,A -85,B 0,C 180,E1 -10930.21,E2 -10930.21} C_VEL
LIN {X 0,Y 403.596,Z 448.199,A -85,B 0,C 180,E1 -10932.007,E2 -10932.007} C_VEL
LIN {X 0,Y 413.32,Z 391.687,A -85,B 0,C 180,E1 -10933.887,E2 -10933.887} C_VEL
LIN {X 0,Y 417.462,Z 370.843,A -85,B 0,C 180,E1 -10934.603,E2 -10934.603} C_VEL
LIN {X 0,Y 416.625,Z 368.637,A -85,B 0,C 180,E1 -10936.053,E2 -10936.053} C_VEL
LIN {X 0,Y 416.23,Z 370.282,A -85,B 0,C 180,E1 -10937.648,E2 -10937.648} C_VEL
LIN {X 0,Y 416.609,Z 374.396,A -85,B 0,C 180,E1 -10939.114,E2 -10939.114} C_VEL
LIN {X 0,Y 416.295,Z 377.115,A -85,B 0,C 180,E1 -10939.375,E2 -10939.375} C_VEL
LIN {X 0,Y 414.994,Z 386.565,A -85,B 0,C 180,E1 -10940.036,E2 -10940.036} C_VEL
LIN {X 0,Y 402.614,Z 455.585,A -85,B 0,C 180,E1 -10942.378,E2 -10942.378} C_VEL
LIN {X 0,Y 393.658,Z 518.567,A -85,B 0,C 180,E1 -10944.524,E2 -10944.524} C_VEL
LIN {X 0,Y 387.47,Z 572.808,A -85,B 0,C 180,E1 -10946.359,E2 -10946.359} C_VEL
LIN {X 0,Y 384.736,Z 593.941,A -85,B 0,C 180,E1 -10947.368,E2 -10947.368} C_VEL
LIN {X 0,Y 381.83,Z 613.98,A -85,B 0,C 180,E1 -10948.614,E2 -10948.614} C_VEL
LIN {X 0,Y 378.704,Z 633.508,A -85,B 0,C 180,E1 -10950.154,E2 -10950.154} C_VEL
LIN {X 0,Y 375.638,Z 651.411,A -85,B 0,C 180,E1 -10951.893,E2 -10951.893} C_VEL
LIN {X 0,Y 372.601,Z 668.27,A -85,B 0,C 180,E1 -10953.891,E2 -10953.891} C_VEL
LIN {X 0,Y 369.779,Z 683.433,A -85,B 0,C 180,E1 -10956.072,E2 -10956.072} C_VEL
LIN {X 0,Y 367.393,Z 696.148,A -85,B 0,C 180,E1 -10958.277,E2 -10958.277} C_VEL
LIN {X 0,Y 365.287,Z 707.58,A -85,B 0,C 180,E1 -10960.659,E2 -10960.659} C_VEL
LIN {X 0,Y 363.518,Z 717.679,A -85,B 0,C 180,E1 -10963.214,E2 -10963.214} C_VEL
LIN {X 0,Y 362.121,Z 726.367,A -85,B 0,C 180,E1 -10965.938,E2 -10965.938} C_VEL
LIN {X 0,Y 361.126,Z 733.552,A -85,B 0,C 180,E1 -10968.825,E2 -10968.825} C_VEL
LIN {X 0,Y 360.532,Z 738.865,A -85,B 0,C 180,E1 -10971.709,E2 -10971.709} C_VEL
LIN {X 0,Y 360.229,Z 742.445,A -85,B 0,C 180,E1 -10974.585,E2 -10974.585} C_VEL
LIN {X 0,Y 360.095,Z 744.439,A -85,B 0,C 180,E1 -10977.614,E2 -10977.614} C_VEL
LIN {X 0,Y 360.063,Z 744.673,A -85,B 0,C 180,E1 -10980.478,E2 -10980.478} C_VEL
LIN {X 0,Y 360.078,Z 743.299,A -85,B 0,C 180,E1 -10983.344,E2 -10983.344} C_VEL
LIN {X 0,Y 360.185,Z 740.297,A -85,B 0,C 180,E1 -10986.216,E2 -10986.216} C_VEL
LIN {X 0,Y 360.473,Z 735.589,A -85,B 0,C 180,E1 -10989.097,E2 -10989.097} C_VEL
LIN {X 0,Y 361.018,Z 729.481,A -85,B 0,C 180,E1 -10991.827,E2 -10991.827} C_VEL
LIN {X 0,Y 361.907,Z 721.59,A -85,B 0,C 180,E1 -10994.562,E2 -10994.562} C_VEL
LIN {X 0,Y 363.22,Z 711.678,A -85,B 0,C 180,E1 -10997.296,E2 -10997.296} C_VEL
LIN {X 0,Y 364.906,Z 700.221,A -85,B 0,C 180,E1 -10999.863,E2 -10999.863} C_VEL
LIN {X 0,Y 366.92,Z 687.23,A -85,B 0,C 180,E1 -11002.259,E2 -11002.259} C_VEL
LIN {X 0,Y 369.206,Z 672.655,A -85,B 0,C 180,E1 -11004.479,E2 -11004.479} C_VEL
LIN {X 0,Y 371.695,Z 656.362,A -85,B 0,C 180,E1 -11006.523,E2 -11006.523} C_VEL
LIN {X 0,Y 374.101,Z 639.723,A -85,B 0,C 180,E1 -11008.234,E2 -11008.234} C_VEL
LIN {X 0,Y 376.392,Z 622.31,A -85,B 0,C 180,E1 -11009.696,E2 -11009.696} C_VEL
LIN {X 0,Y 378.516,Z 604.11,A -85,B 0,C 180,E1 -11010.916,E2 -11010.916} C_VEL
LIN {X 0,Y 380.423,Z 584.401,A -85,B 0,C 180,E1 -11011.935,E2 -11011.935} C_VEL
LIN {X 0,Y 381.947,Z 564.641,A -85,B 0,C 180,E1 -11012.668,E2 -11012.668} C_VEL
LIN {X 0,Y 384.109,Z 518.749,A -85,B 0,C 180,E1 -11013.775,E2 -11013.775} C_VEL
LIN {X 0,Y 390.905,Z 378.386,A -85,B 0,C 180,E1 -11017.055,E2 -11017.055} C_VEL
LIN {X 0,Y 387.233,Z 352.342,A -85,B 0,C 180,E1 -11018.193,E2 -11018.193} C_VEL
LIN {X 0,Y 380.321,Z 338.936,A -85,B 0,C 180,E1 -11019.381,E2 -11019.381} C_VEL
LIN {X 0,Y 372.972,Z 319.156,A -85,B 0,C 180,E1 -11022.843,E2 -11022.843} C_VEL
LIN {X 0,Y 365.795,Z 301.475,A -85,B 0,C 180,E1 -11026.246,E2 -11026.246} C_VEL
LIN {X 0,Y 361.828,Z 291.608,A -85,B 0,C 180,E1 -11028.321,E2 -11028.321} C_VEL
LIN {X 0,Y 361.805,Z 291.418,A -85,B 0,C 180,E1 -11032.48,E2 -11032.48} C_VEL
LIN {X 0,Y 361.803,Z 291.417,A -85,B 0,C 180,E1 -11036.635,E2 -11036.635} C_VEL
LIN {X 0,Y 361.793,Z 291.394,A -85,B 0,C 180,E1 -11040.713,E2 -11040.713} C_VEL
LIN {X 0,Y 361.781,Z 291.399,A -85,B 0,C 180,E1 -11044.809,E2 -11044.809} C_VEL
LIN {X 0,Y 361.849,Z 291.658,A -85,B 0,C 180,E1 -11047.882,E2 -11047.882} C_VEL
LIN {X 0,Y 364.914,Z 298.892,A -85,B 0,C 180,E1 -11049.123,E2 -11049.123} C_VEL
LIN {X 0,Y 372.715,Z 317.86,A -85,B 0,C 180,E1 -11052.11,E2 -11052.11} C_VEL
LIN {X 0,Y 379.259,Z 336.41,A -85,B 0,C 180,E1 -11054.778,E2 -11054.778} C_VEL
LIN {X 0,Y 381.599,Z 344.037,A -85,B 0,C 180,E1 -11055.808,E2 -11055.808} C_VEL
LIN {X 0,Y 378.865,Z 384.794,A -85,B 0,C 180,E1 -11059.722,E2 -11059.722} C_VEL
LIN {X 0,Y 376.074,Z 426.012,A -85,B 0,C 180,E1 -11063.664,E2 -11063.664} C_VEL
LIN {X 0,Y 375.3,Z 438.327,A -85,B 0,C 180,E1 -11064.849,E2 -11064.849} C_VEL
LIN {X 0,Y 373.99,Z 445.018,A -85,B 0,C 180,E1 -11065.416,E2 -11065.416} C_VEL
LIN {X 0,Y 367.132,Z 463.306,A -85,B 0,C 180,E1 -11066.716,E2 -11066.716} C_VEL
LIN {X 0,Y 366.041,Z 469.044,A -85,B 0,C 180,E1 -11067.221,E2 -11067.221} C_VEL
LIN {X 0,Y 365.34,Z 480.845,A -85,B 0,C 180,E1 -11068.322,E2 -11068.322} C_VEL
LIN {X 0,Y 367.274,Z 500.091,A -85,B 0,C 180,E1 -11068.887,E2 -11068.887} C_VEL
LIN {X 0,Y 364.343,Z 624.371,A -85,B 0,C 180,E1 -11071.399,E2 -11071.399} C_VEL
LIN {X 0,Y 363.607,Z 640.39,A -85,B 0,C 180,E1 -11072.011,E2 -11072.011} C_VEL
LIN {X 0,Y 362.484,Z 656.498,A -85,B 0,C 180,E1 -11072.931,E2 -11072.931} C_VEL
LIN {X 0,Y 361.159,Z 670.777,A -85,B 0,C 180,E1 -11074.046,E2 -11074.046} C_VEL
LIN {X 0,Y 359.596,Z 684.917,A -85,B 0,C 180,E1 -11075.477,E2 -11075.477} C_VEL
LIN {X 0,Y 358.065,Z 697.249,A -85,B 0,C 180,E1 -11077.056,E2 -11077.056} C_VEL
LIN {X 0,Y 356.414,Z 709.709,A -85,B 0,C 180,E1 -11079.073,E2 -11079.073} C_VEL
LIN {X 0,Y 355.108,Z 719.37,A -85,B 0,C 180,E1 -11081.036,E2 -11081.036} C_VEL
LIN {X 0,Y 353.909,Z 728.488,A -85,B 0,C 180,E1 -11083.393,E2 -11083.393} C_VEL
LIN {X 0,Y 353.071,Z 735.573,A -85,B 0,C 180,E1 -11085.773,E2 -11085.773} C_VEL
LIN {X 0,Y 352.513,Z 741.144,A -85,B 0,C 180,E1 -11088.349,E2 -11088.349} C_VEL
LIN {X 0,Y 352.233,Z 744.901,A -85,B 0,C 180,E1 -11090.955,E2 -11090.955} C_VEL
LIN {X 0,Y 352.125,Z 746.856,A -85,B 0,C 180,E1 -11093.599,E2 -11093.599} C_VEL
LIN {X 0,Y 352.13,Z 747.086,A -85,B 0,C 180,E1 -11096.29,E2 -11096.29} C_VEL
LIN {X 0,Y 352.235,Z 745.556,A -85,B 0,C 180,E1 -11098.851,E2 -11098.851} C_VEL
LIN {X 0,Y 352.521,Z 742.31,A -85,B 0,C 180,E1 -11101.456,E2 -11101.456} C_VEL
LIN {X 0,Y 353.041,Z 737.486,A -85,B 0,C 180,E1 -11103.919,E2 -11103.919} C_VEL
LIN {X 0,Y 353.901,Z 730.768,A -85,B 0,C 180,E1 -11106.389,E2 -11106.389} C_VEL
LIN {X 0,Y 355.064,Z 722.531,A -85,B 0,C 180,E1 -11108.69,E2 -11108.69} C_VEL
LIN {X 0,Y 356.577,Z 712.182,A -85,B 0,C 180,E1 -11110.937,E2 -11110.937} C_VEL
LIN {X 0,Y 358.152,Z 701.269,A -85,B 0,C 180,E1 -11112.813,E2 -11112.813} C_VEL
LIN {X 0,Y 359.962,Z 687.793,A -85,B 0,C 180,E1 -11114.645,E2 -11114.645} C_VEL
LIN {X 0,Y 361.603,Z 674.011,A -85,B 0,C 180,E1 -11116.107,E2 -11116.107} C_VEL
LIN {X 0,Y 363.109,Z 659.138,A -85,B 0,C 180,E1 -11117.322,E2 -11117.322} C_VEL
LIN {X 0,Y 364.287,Z 643.643,A -85,B 0,C 180,E1 -11118.254,E2 -11118.254} C_VEL
LIN {X 0,Y 365.139,Z 626.953,A -85,B 0,C 180,E1 -11118.937,E2 -11118.937} C_VEL
LIN {X 0,Y 365.879,Z 597.165,A -85,B 0,C 180,E1 -11119.594,E2 -11119.594} C_VEL
LIN {X 0,Y 368.221,Z 497.455,A -85,B 0,C 180,E1 -11121.612,E2 -11121.612} C_VEL
LIN {X 0,Y 366.373,Z 481.041,A -85,B 0,C 180,E1 -11122.164,E2 -11122.164} C_VEL
LIN {X 0,Y 369.311,Z 437.955,A -85,B 0,C 180,E1 -11126.288,E2 -11126.288} C_VEL
LIN {X 0,Y 372.235,Z 396.103,A -85,B 0,C 180,E1 -11130.291,E2 -11130.291} C_VEL
LIN {X 0,Y 374.913,Z 355.379,A -85,B 0,C 180,E1 -11134.148,E2 -11134.148} C_VEL
LIN {X 0,Y 375.452,Z 346.139,A -85,B 0,C 180,E1 -11135.032,E2 -11135.032} C_VEL
LIN {X 0,Y 370.078,Z 329.501,A -85,B 0,C 180,E1 -11137.439,E2 -11137.439} C_VEL
LIN {X 0,Y 363.906,Z 314.09,A -85,B 0,C 180,E1 -11139.912,E2 -11139.912} C_VEL
LIN {X 0,Y 357.873,Z 300.913,A -85,B 0,C 180,E1 -11142.269,E2 -11142.269} C_VEL
LIN {X 0,Y 355.495,Z 296.371,A -85,B 0,C 180,E1 -11143.16,E2 -11143.16} C_VEL
LIN {X 0,Y 353.908,Z 292.857,A -85,B 0,C 180,E1 -11143.88,E2 -11143.88} C_VEL
LIN {X 0,Y 353.868,Z 292.394,A -85,B 0,C 180,E1 -11144.463,E2 -11144.463} C_VEL
LIN {X 0,Y 353.866,Z 292.409,A -85,B 0,C 180,E1 -11148.642,E2 -11148.642} C_VEL
LIN {X 0,Y 353.871,Z 292.405,A -85,B 0,C 180,E1 -11152.858,E2 -11152.858} C_VEL
LIN {X 0,Y 353.854,Z 292.409,A -85,B 0,C 180,E1 -11157.084,E2 -11157.084} C_VEL
LIN {X 0,Y 353.856,Z 292.401,A -85,B 0,C 180,E1 -11161.133,E2 -11161.133} C_VEL
LIN {X 0,Y 353.849,Z 292.408,A -85,B 0,C 180,E1 -11165.35,E2 -11165.35} C_VEL
LIN {X 0,Y 353.847,Z 292.401,A -85,B 0,C 180,E1 -11169.432,E2 -11169.432} C_VEL
LIN {X 0,Y 353.844,Z 292.407,A -85,B 0,C 180,E1 -11173.591,E2 -11173.591} C_VEL
LIN {X 0,Y 353.844,Z 292.409,A -85,B 0,C 180,E1 -11177.783,E2 -11177.783} C_VEL
LIN {X 0,Y 353.839,Z 292.402,A -85,B 0,C 180,E1 -11182.075,E2 -11182.075} C_VEL
LIN {X 0,Y 353.845,Z 292.41,A -85,B 0,C 180,E1 -11186.155,E2 -11186.155} C_VEL
LIN {X 0,Y 353.847,Z 292.405,A -85,B 0,C 180,E1 -11190.196,E2 -11190.196} C_VEL
LIN {X 0,Y 353.85,Z 292.405,A -85,B 0,C 180,E1 -11194.411,E2 -11194.411} C_VEL
LIN {X 0,Y 353.897,Z 292.66,A -85,B 0,C 180,E1 -11197.495,E2 -11197.495} C_VEL
LIN {X 0,Y 357.045,Z 299.971,A -85,B 0,C 180,E1 -11199.056,E2 -11199.056} C_VEL
LIN {X 0,Y 365.164,Z 318.697,A -85,B 0,C 180,E1 -11202.662,E2 -11202.662} C_VEL
LIN {X 0,Y 366.884,Z 322.019,A -85,B 0,C 180,E1 -11203.106,E2 -11203.106} C_VEL
LIN {X 0,Y 382.509,Z 349.027,A -85,B 0,C 180,E1 -11205.823,E2 -11205.823} C_VEL
LIN {X 0,Y 389.851,Z 362.656,A -85,B 0,C 180,E1 -11207.036,E2 -11207.036} C_VEL
LIN {X 0,Y 379.031,Z 577.128,A -85,B 0,C 180,E1 -11211.987,E2 -11211.987} C_VEL
LIN {X 0,Y 377.266,Z 598.585,A -85,B 0,C 180,E1 -11212.748,E2 -11212.748} C_VEL
LIN {X 0,Y 375.037,Z 619.279,A -85,B 0,C 180,E1 -11213.761,E2 -11213.761} C_VEL
LIN {X 0,Y 372.468,Z 639.496,A -85,B 0,C 180,E1 -11215.054,E2 -11215.054} C_VEL
LIN {X 0,Y 369.666,Z 658.814,A -85,B 0,C 180,E1 -11216.607,E2 -11216.607} C_VEL
LIN {X 0,Y 366.714,Z 677.354,A -85,B 0,C 180,E1 -11218.435,E2 -11218.435} C_VEL
LIN {X 0,Y 363.865,Z 694.194,A -85,B 0,C 180,E1 -11220.448,E2 -11220.448} C_VEL
LIN {X 0,Y 361.19,Z 709.59,A -85,B 0,C 180,E1 -11222.646,E2 -11222.646} C_VEL
LIN {X 0,Y 358.686,Z 724.094,A -85,B 0,C 180,E1 -11225.109,E2 -11225.109} C_VEL
LIN {X 0,Y 356.53,Z 737.136,A -85,B 0,C 180,E1 -11227.755,E2 -11227.755} C_VEL
LIN {X 0,Y 354.787,Z 748.722,A -85,B 0,C 180,E1 -11230.579,E2 -11230.579} C_VEL
LIN {X 0,Y 353.51,Z 758.583,A -85,B 0,C 180,E1 -11233.498,E2 -11233.498} C_VEL
LIN {X 0,Y 352.651,Z 766.912,A -85,B 0,C 180,E1 -11236.558,E2 -11236.558} C_VEL
LIN {X 0,Y 352.202,Z 773.508,A -85,B 0,C 180,E1 -11239.699,E2 -11239.699} C_VEL
LIN {X 0,Y 352.042,Z 778.044,A -85,B 0,C 180,E1 -11242.659,E2 -11242.659} C_VEL
LIN {X 0,Y 352.043,Z 781.185,A -85,B 0,C 180,E1 -11245.767,E2 -11245.767} C_VEL
LIN {X 0,Y 352.064,Z 782.659,A -85,B 0,C 180,E1 -11248.7,E2 -11248.7} C_VEL
LIN {X 0,Y 352.063,Z 782.558,A -85,B 0,C 180,E1 -11251.629,E2 -11251.629} C_VEL
LIN {X 0,Y 352.03,Z 780.87,A -85,B 0,C 180,E1 -11254.726,E2 -11254.726} C_VEL
LIN {X 0,Y 352.059,Z 777.546,A -85,B 0,C 180,E1 -11257.837,E2 -11257.837} C_VEL
LIN {X 0,Y 352.265,Z 772.518,A -85,B 0,C 180,E1 -11260.964,E2 -11260.964} C_VEL
LIN {X 0,Y 352.8,Z 765.61,A -85,B 0,C 180,E1 -11264.108,E2 -11264.108} C_VEL
LIN {X 0,Y 353.738,Z 757.245,A -85,B 0,C 180,E1 -11267.097,E2 -11267.097} C_VEL
LIN {X 0,Y 355.188,Z 746.947,A -85,B 0,C 180,E1 -11270.088,E2 -11270.088} C_VEL
LIN {X 0,Y 357.225,Z 734.416,A -85,B 0,C 180,E1 -11273.071,E2 -11273.071} C_VEL
LIN {X 0,Y 359.635,Z 720.906,A -85,B 0,C 180,E1 -11275.739,E2 -11275.739} C_VEL
LIN {X 0,Y 362.434,Z 705.823,A -85,B 0,C 180,E1 -11278.239,E2 -11278.239} C_VEL
LIN {X 0,Y 365.622,Z 688.919,A -85,B 0,C 180,E1 -11280.575,E2 -11280.575} C_VEL
LIN {X 0,Y 368.931,Z 671.004,A -85,B 0,C 180,E1 -11282.639,E2 -11282.639} C_VEL
LIN {X 0,Y 372.339,Z 651.793,A -85,B 0,C 180,E1 -11284.473,E2 -11284.473} C_VEL
LIN {X 0,Y 375.847,Z 630.869,A -85,B 0,C 180,E1 -11286.099,E2 -11286.099} C_VEL
LIN {X 0,Y 379.16,Z 609.366,A -85,B 0,C 180,E1 -11287.435,E2 -11287.435} C_VEL
LIN {X 0,Y 382.265,Z 587.239,A -85,B 0,C 180,E1 -11288.49,E2 -11288.49} C_VEL
LIN {X 0,Y 385.075,Z 563.095,A -85,B 0,C 180,E1 -11289.344,E2 -11289.344} C_VEL
LIN {X 0,Y 391.254,Z 508.421,A -85,B 0,C 180,E1 -11291.055,E2 -11291.055} C_VEL
LIN {X 0,Y 399.432,Z 454.052,A -85,B 0,C 180,E1 -11292.87,E2 -11292.87} C_VEL
LIN {X 0,Y 409.983,Z 399.107,A -85,B 0,C 180,E1 -11294.742,E2 -11294.742} C_VEL
LIN {X 0,Y 414.784,Z 377.197,A -85,B 0,C 180,E1 -11295.499,E2 -11295.499} C_VEL
LIN {X 0,Y 414.542,Z 376.403,A -85,B 0,C 180,E1 -11296.193,E2 -11296.193} C_VEL
LIN {X 0,Y 414.117,Z 378.19,A -85,B 0,C 180,E1 -11297.569,E2 -11297.569} C_VEL
LIN {X 0,Y 414.089,Z 380.818,A -85,B 0,C 180,E1 -11298.445,E2 -11298.445} C_VEL
LIN {X 0,Y 412.662,Z 388.813,A -85,B 0,C 180,E1 -11299.015,E2 -11299.015} C_VEL
LIN {X 0,Y 398.922,Z 457.859,A -85,B 0,C 180,E1 -11301.402,E2 -11301.402} C_VEL
LIN {X 0,Y 388.944,Z 520.401,A -85,B 0,C 180,E1 -11303.605,E2 -11303.605} C_VEL
LIN {X 0,Y 382.044,Z 573.666,A -85,B 0,C 180,E1 -11305.493,E2 -11305.493} C_VEL
LIN {X 0,Y 378.992,Z 594.737,A -85,B 0,C 180,E1 -11306.538,E2 -11306.538} C_VEL
LIN {X 0,Y 375.73,Z 615.001,A -85,B 0,C 180,E1 -11307.845,E2 -11307.845} C_VEL
LIN {X 0,Y 372.349,Z 634.296,A -85,B 0,C 180,E1 -11309.413,E2 -11309.413} C_VEL
LIN {X 0,Y 368.925,Z 652.617,A -85,B 0,C 180,E1 -11311.246,E2 -11311.246} C_VEL
LIN {X 0,Y 365.683,Z 669.205,A -85,B 0,C 180,E1 -11313.269,E2 -11313.269} C_VEL
LIN {X 0,Y 362.675,Z 684.156,A -85,B 0,C 180,E1 -11315.477,E2 -11315.477} C_VEL
LIN {X 0,Y 360.016,Z 697.247,A -85,B 0,C 180,E1 -11317.809,E2 -11317.809} C_VEL
LIN {X 0,Y 357.627,Z 709.237,A -85,B 0,C 180,E1 -11320.398,E2 -11320.398} C_VEL
LIN {X 0,Y 355.652,Z 719.675,A -85,B 0,C 180,E1 -11323.168,E2 -11323.168} C_VEL
LIN {X 0,Y 354.138,Z 728.499,A -85,B 0,C 180,E1 -11326.115,E2 -11326.115} C_VEL
LIN {X 0,Y 353.133,Z 735.287,A -85,B 0,C 180,E1 -11329.065,E2 -11329.065} C_VEL
LIN {X 0,Y 352.533,Z 740.238,A -85,B 0,C 180,E1 -11332.012,E2 -11332.012} C_VEL
LIN {X 0,Y 352.221,Z 743.615,A -85,B 0,C 180,E1 -11335.115,E2 -11335.115} C_VEL
LIN {X 0,Y 352.102,Z 745.165,A -85,B 0,C 180,E1 -11338.211,E2 -11338.211} C_VEL
LIN {X 0,Y 352.078,Z 744.964,A -85,B 0,C 180,E1 -11341.14,E2 -11341.14} C_VEL
LIN {X 0,Y 352.101,Z 743.142,A -85,B 0,C 180,E1 -11344.072,E2 -11344.072} C_VEL
LIN {X 0,Y 352.254,Z 739.671,A -85,B 0,C 180,E1 -11347.011,E2 -11347.011} C_VEL
LIN {X 0,Y 352.635,Z 734.466,A -85,B 0,C 180,E1 -11349.961,E2 -11349.961} C_VEL
LIN {X 0,Y 353.289,Z 727.831,A -85,B 0,C 180,E1 -11352.754,E2 -11352.754} C_VEL
LIN {X 0,Y 354.339,Z 719.363,A -85,B 0,C 180,E1 -11355.55,E2 -11355.55} C_VEL
LIN {X 0,Y 355.767,Z 709.37,A -85,B 0,C 180,E1 -11358.205,E2 -11358.205} C_VEL
LIN {X 0,Y 357.628,Z 697.449,A -85,B 0,C 180,E1 -11360.798,E2 -11360.798} C_VEL
LIN {X 0,Y 359.767,Z 684.297,A -85,B 0,C 180,E1 -11363.158,E2 -11363.158} C_VEL
LIN {X 0,Y 362.151,Z 669.647,A -85,B 0,C 180,E1 -11365.337,E2 -11365.337} C_VEL
LIN {X 0,Y 364.723,Z 653.29,A -85,B 0,C 180,E1 -11367.347,E2 -11367.347} C_VEL
LIN {X 0,Y 367.283,Z 635.924,A -85,B 0,C 180,E1 -11369.087,E2 -11369.087} C_VEL
LIN {X 0,Y 369.705,Z 617.67,A -85,B 0,C 180,E1 -11370.561,E2 -11370.561} C_VEL
LIN {X 0,Y 371.868,Z 598.902,A -85,B 0,C 180,E1 -11371.758,E2 -11371.758} C_VEL
LIN {X 0,Y 373.752,Z 579.176,A -85,B 0,C 180,E1 -11372.711,E2 -11372.711} C_VEL
LIN {X 0,Y 375.216,Z 558.965,A -85,B 0,C 180,E1 -11373.398,E2 -11373.398} C_VEL
LIN {X 0,Y 384.268,Z 379.693,A -85,B 0,C 180,E1 -11377.696,E2 -11377.696} C_VEL
LIN {X 0,Y 380.901,Z 355.727,A -85,B 0,C 180,E1 -11378.773,E2 -11378.773} C_VEL
LIN {X 0,Y 372.105,Z 338.803,A -85,B 0,C 180,E1 -11380.328,E2 -11380.328} C_VEL
LIN {X 0,Y 364.897,Z 319.706,A -85,B 0,C 180,E1 -11383.777,E2 -11383.777} C_VEL
LIN {X 0,Y 358.197,Z 303.093,A -85,B 0,C 180,E1 -11387.069,E2 -11387.069} C_VEL
LIN {X 0,Y 353.898,Z 292.602,A -85,B 0,C 180,E1 -11389.346,E2 -11389.346} C_VEL
LIN {X 0,Y 353.864,Z 292.405,A -85,B 0,C 180,E1 -11393.401,E2 -11393.401} C_VEL
LIN {X 0,Y 353.868,Z 292.405,A -85,B 0,C 180,E1 -11397.655,E2 -11397.655} C_VEL
LIN {X 0,Y 353.878,Z 292.389,A -85,B 0,C 180,E1 -11401.844,E2 -11401.844} C_VEL
LIN {X 0,Y 353.868,Z 292.392,A -85,B 0,C 180,E1 -11406.167,E2 -11406.167} C_VEL
LIN {X 0,Y 353.881,Z 292.683,A -85,B 0,C 180,E1 -11406.918,E2 -11406.918} C_VEL
LIN {X 0,Y 355.345,Z 296.146,A -85,B 0,C 180,E1 -11407.568,E2 -11407.568} C_VEL
LIN {X 0,Y 363,Z 313.908,A -85,B 0,C 180,E1 -11410.53,E2 -11410.53} C_VEL
LIN {X 0,Y 369.965,Z 332.505,A -85,B 0,C 180,E1 -11413.352,E2 -11413.352} C_VEL
LIN {X 0,Y 374.563,Z 347.008,A -85,B 0,C 180,E1 -11415.387,E2 -11415.387} C_VEL
LIN {X 0,Y 371.681,Z 388.244,A -85,B 0,C 180,E1 -11419.38,E2 -11419.38} C_VEL
LIN {X 0,Y 368.71,Z 429.481,A -85,B 0,C 180,E1 -11423.38,E2 -11423.38} C_VEL
LIN {X 0,Y 366.041,Z 469.044,A -85,B 0,C 180,E1 -11427.221,E2 -11427.221} C_VEL
LIN {X 0,Y 364.887,Z 473.69,A -85,B 0,C 180,E1 -11427.568,E2 -11427.568} C_VEL
LIN {X 0,Y 360.9,Z 482.615,A -85,B 0,C 180,E1 -11427.88,E2 -11427.88} C_VEL
LIN {X 0,Y 359.261,Z 488.42,A -85,B 0,C 180,E1 -11428.008,E2 -11428.008} C_VEL
LIN {X 0,Y 359.22,Z 491.389,A -85,B 0,C 180,E1 -11428.089,E2 -11428.089} C_VEL
LIN {X 0,Y 360.012,Z 501.251,A -85,B 0,C 180,E1 -11428.37,E2 -11428.37} C_VEL
LIN {X 0,Y 356.963,Z 624.676,A -85,B 0,C 180,E1 -11430.911,E2 -11430.911} C_VEL
LIN {X 0,Y 356.194,Z 640.757,A -85,B 0,C 180,E1 -11431.536,E2 -11431.536} C_VEL
LIN {X 0,Y 355.087,Z 656.045,A -85,B 0,C 180,E1 -11432.419,E2 -11432.419} C_VEL
LIN {X 0,Y 353.694,Z 670.658,A -85,B 0,C 180,E1 -11433.564,E2 -11433.564} C_VEL
LIN {X 0,Y 352.026,Z 685.133,A -85,B 0,C 180,E1 -11435.05,E2 -11435.05} C_VEL
LIN {X 0,Y 350.364,Z 697.92,A -85,B 0,C 180,E1 -11436.722,E2 -11436.722} C_VEL
LIN {X 0,Y 348.671,Z 710.11,A -85,B 0,C 180,E1 -11438.74,E2 -11438.74} C_VEL
LIN {X 0,Y 347.272,Z 719.928,A -85,B 0,C 180,E1 -11440.784,E2 -11440.784} C_VEL
LIN {X 0,Y 346.014,Z 729.02,A -85,B 0,C 180,E1 -11443.194,E2 -11443.194} C_VEL
LIN {X 0,Y 345.13,Z 736.064,A -85,B 0,C 180,E1 -11445.628,E2 -11445.628} C_VEL
LIN {X 0,Y 344.524,Z 741.813,A -85,B 0,C 180,E1 -11448.375,E2 -11448.375} C_VEL
LIN {X 0,Y 344.246,Z 745.333,A -85,B 0,C 180,E1 -11450.929,E2 -11450.929} C_VEL
LIN {X 0,Y 344.133,Z 747.32,A -85,B 0,C 180,E1 -11453.762,E2 -11453.762} C_VEL
LIN {X 0,Y 344.142,Z 747.461,A -85,B 0,C 180,E1 -11456.39,E2 -11456.39} C_VEL
LIN {X 0,Y 344.275,Z 745.73,A -85,B 0,C 180,E1 -11459.201,E2 -11459.201} C_VEL
LIN {X 0,Y 344.607,Z 742.318,A -85,B 0,C 180,E1 -11461.872,E2 -11461.872} C_VEL
LIN {X 0,Y 345.259,Z 736.861,A -85,B 0,C 180,E1 -11464.581,E2 -11464.581} C_VEL
LIN {X 0,Y 346.168,Z 730.414,A -85,B 0,C 180,E1 -11466.923,E2 -11466.923} C_VEL
LIN {X 0,Y 347.447,Z 721.905,A -85,B 0,C 180,E1 -11469.276,E2 -11469.276} C_VEL
LIN {X 0,Y 349.057,Z 711.622,A -85,B 0,C 180,E1 -11471.51,E2 -11471.51} C_VEL
LIN {X 0,Y 350.826,Z 699.81,A -85,B 0,C 180,E1 -11473.517,E2 -11473.517} C_VEL
LIN {X 0,Y 352.53,Z 687.765,A -85,B 0,C 180,E1 -11475.155,E2 -11475.155} C_VEL
LIN {X 0,Y 354.266,Z 673.752,A -85,B 0,C 180,E1 -11476.652,E2 -11476.652} C_VEL
LIN {X 0,Y 355.842,Z 658.826,A -85,B 0,C 180,E1 -11477.881,E2 -11477.881} C_VEL
LIN {X 0,Y 357.082,Z 642.927,A -85,B 0,C 180,E1 -11478.834,E2 -11478.834} C_VEL
LIN {X 0,Y 357.937,Z 626.53,A -85,B 0,C 180,E1 -11479.501,E2 -11479.501} C_VEL
LIN {X 0,Y 359.191,Z 577.723,A -85,B 0,C 180,E1 -11480.552,E2 -11480.552} C_VEL
LIN {X 0,Y 361.15,Z 498.272,A -85,B 0,C 180,E1 -11482.194,E2 -11482.194} C_VEL
LIN {X 0,Y 359.27,Z 481.145,A -85,B 0,C 180,E1 -11482.798,E2 -11482.798} C_VEL
LIN {X 0,Y 362.404,Z 437.841,A -85,B 0,C 180,E1 -11487.001,E2 -11487.001} C_VEL
LIN {X 0,Y 365.258,Z 398.895,A -85,B 0,C 180,E1 -11490.758,E2 -11490.758} C_VEL
LIN {X 0,Y 368.005,Z 360.056,A -85,B 0,C 180,E1 -11494.482,E2 -11494.482} C_VEL
LIN {X 0,Y 368.62,Z 349.005,A -85,B 0,C 180,E1 -11495.565,E2 -11495.565} C_VEL
LIN {X 0,Y 363.275,Z 332.476,A -85,B 0,C 180,E1 -11498.017,E2 -11498.017} C_VEL
LIN {X 0,Y 357.268,Z 317.255,A -85,B 0,C 180,E1 -11500.546,E2 -11500.546} C_VEL
LIN {X 0,Y 350.123,Z 302.104,A -85,B 0,C 180,E1 -11503.406,E2 -11503.406} C_VEL
LIN {X 0,Y 347.358,Z 297.043,A -85,B 0,C 180,E1 -11504.472,E2 -11504.472} C_VEL
LIN {X 0,Y 345.947,Z 293.7,A -85,B 0,C 180,E1 -11505.222,E2 -11505.222} C_VEL
LIN {X 0,Y 345.917,Z 293.398,A -85,B 0,C 180,E1 -11506.97,E2 -11506.97} C_VEL
LIN {X 0,Y 345.908,Z 293.395,A -85,B 0,C 180,E1 -11511.187,E2 -11511.187} C_VEL
LIN {X 0,Y 345.904,Z 293.396,A -85,B 0,C 180,E1 -11515.357,E2 -11515.357} C_VEL
LIN {X 0,Y 345.899,Z 293.399,A -85,B 0,C 180,E1 -11519.668,E2 -11519.668} C_VEL
LIN {X 0,Y 345.901,Z 293.392,A -85,B 0,C 180,E1 -11523.977,E2 -11523.977} C_VEL
LIN {X 0,Y 345.904,Z 293.398,A -85,B 0,C 180,E1 -11528.142,E2 -11528.142} C_VEL
LIN {X 0,Y 345.911,Z 293.391,A -85,B 0,C 180,E1 -11532.35,E2 -11532.35} C_VEL
LIN {X 0,Y 345.917,Z 293.39,A -85,B 0,C 180,E1 -11536.455,E2 -11536.455} C_VEL
LIN {X 0,Y 345.926,Z 293.396,A -85,B 0,C 180,E1 -11540.647,E2 -11540.647} C_VEL
LIN {X 0,Y 345.928,Z 293.39,A -85,B 0,C 180,E1 -11544.834,E2 -11544.834} C_VEL
LIN {X 0,Y 345.94,Z 293.391,A -85,B 0,C 180,E1 -11549.049,E2 -11549.049} C_VEL
LIN {X 0,Y 345.926,Z 293.395,A -85,B 0,C 180,E1 -11553.355,E2 -11553.355} C_VEL
LIN {X 0,Y 345.947,Z 293.653,A -85,B 0,C 180,E1 -11556.377,E2 -11556.377} C_VEL
LIN {X 0,Y 349.101,Z 300.999,A -85,B 0,C 180,E1 -11558.008,E2 -11558.008} C_VEL
LIN {X 0,Y 356.998,Z 319.001,A -85,B 0,C 180,E1 -11561.604,E2 -11561.604} C_VEL
LIN {X 0,Y 358.404,Z 321.821,A -85,B 0,C 180,E1 -11562.004,E2 -11562.004} C_VEL
LIN {X 0,Y 373.606,Z 347.823,A -85,B 0,C 180,E1 -11564.763,E2 -11564.763} C_VEL
LIN {X 0,Y 383.238,Z 365.509,A -85,B 0,C 180,E1 -11566.399,E2 -11566.399} C_VEL
LIN {X 0,Y 372.019,Z 577.042,A -85,B 0,C 180,E1 -11571.397,E2 -11571.397} C_VEL
LIN {X 0,Y 370.171,Z 598.602,A -85,B 0,C 180,E1 -11572.179,E2 -11572.179} C_VEL
LIN {X 0,Y 367.915,Z 618.856,A -85,B 0,C 180,E1 -11573.187,E2 -11573.187} C_VEL
LIN {X 0,Y 365.208,Z 639.397,A -85,B 0,C 180,E1 -11574.523,E2 -11574.523} C_VEL
LIN {X 0,Y 362.281,Z 658.87,A -85,B 0,C 180,E1 -11576.12,E2 -11576.12} C_VEL
LIN {X 0,Y 359.223,Z 677.349,A -85,B 0,C 180,E1 -11577.981,E2 -11577.981} C_VEL
LIN {X 0,Y 356.067,Z 695.384,A -85,B 0,C 180,E1 -11580.191,E2 -11580.191} C_VEL
LIN {X 0,Y 353.131,Z 711.686,A -85,B 0,C 180,E1 -11582.609,E2 -11582.609} C_VEL
LIN {X 0,Y 350.53,Z 726.275,A -85,B 0,C 180,E1 -11585.212,E2 -11585.212} C_VEL
LIN {X 0,Y 348.314,Z 739.285,A -85,B 0,C 180,E1 -11588,E2 -11588} C_VEL
LIN {X 0,Y 346.642,Z 750.137,A -85,B 0,C 180,E1 -11590.805,E2 -11590.805} C_VEL
LIN {X 0,Y 345.37,Z 759.868,A -85,B 0,C 180,E1 -11593.866,E2 -11593.866} C_VEL
LIN {X 0,Y 344.543,Z 768.036,A -85,B 0,C 180,E1 -11597.09,E2 -11597.09} C_VEL
LIN {X 0,Y 344.17,Z 773.995,A -85,B 0,C 180,E1 -11600.133,E2 -11600.133} C_VEL
LIN {X 0,Y 344.051,Z 778.52,A -85,B 0,C 180,E1 -11603.326,E2 -11603.326} C_VEL
LIN {X 0,Y 344.057,Z 781.236,A -85,B 0,C 180,E1 -11606.503,E2 -11606.503} C_VEL
LIN {X 0,Y 344.083,Z 782.274,A -85,B 0,C 180,E1 -11609.502,E2 -11609.502} C_VEL
LIN {X 0,Y 344.063,Z 781.868,A -85,B 0,C 180,E1 -11612.5,E2 -11612.5} C_VEL
LIN {X 0,Y 344.03,Z 779.915,A -85,B 0,C 180,E1 -11615.505,E2 -11615.505} C_VEL
LIN {X 0,Y 344.093,Z 776.22,A -85,B 0,C 180,E1 -11618.692,E2 -11618.692} C_VEL
LIN {X 0,Y 344.378,Z 770.757,A -85,B 0,C 180,E1 -11621.922,E2 -11621.922} C_VEL
LIN {X 0,Y 345.064,Z 763.554,A -85,B 0,C 180,E1 -11625.118,E2 -11625.118} C_VEL
LIN {X 0,Y 346.199,Z 754.865,A -85,B 0,C 180,E1 -11628.176,E2 -11628.176} C_VEL
LIN {X 0,Y 347.906,Z 744.129,A -85,B 0,C 180,E1 -11631.232,E2 -11631.232} C_VEL
LIN {X 0,Y 350.105,Z 731.892,A -85,B 0,C 180,E1 -11634.105,E2 -11634.105} C_VEL
LIN {X 0,Y 352.759,Z 718.215,A -85,B 0,C 180,E1 -11636.788,E2 -11636.788} C_VEL
LIN {X 0,Y 355.919,Z 702.579,A -85,B 0,C 180,E1 -11639.356,E2 -11639.356} C_VEL
LIN {X 0,Y 359.23,Z 686.232,A -85,B 0,C 180,E1 -11641.604,E2 -11641.604} C_VEL
LIN {X 0,Y 362.896,Z 667.84,A -85,B 0,C 180,E1 -11643.715,E2 -11643.715} C_VEL
LIN {X 0,Y 366.559,Z 648.799,A -85,B 0,C 180,E1 -11645.522,E2 -11645.522} C_VEL
LIN {X 0,Y 370.291,Z 628.255,A -85,B 0,C 180,E1 -11647.122,E2 -11647.122} C_VEL
LIN {X 0,Y 373.879,Z 607.143,A -85,B 0,C 180,E1 -11648.437,E2 -11648.437} C_VEL
LIN {X 0,Y 377.388,Z 584.513,A -85,B 0,C 180,E1 -11649.526,E2 -11649.526} C_VEL
LIN {X 0,Y 380.743,Z 558.283,A -85,B 0,C 180,E1 -11650.453,E2 -11650.453} C_VEL
LIN {X 0,Y 387.733,Z 506.206,A -85,B 0,C 180,E1 -11652.173,E2 -11652.173} C_VEL
LIN {X 0,Y 396.994,Z 453.329,A -85,B 0,C 180,E1 -11654.001,E2 -11654.001} C_VEL
LIN {X 0,Y 409.103,Z 397.946,A -85,B 0,C 180,E1 -11655.911,E2 -11655.911} C_VEL
LIN {X 0,Y 412.398,Z 384.444,A -85,B 0,C 180,E1 -11656.363,E2 -11656.363} C_VEL
LIN {X 0,Y 412.031,Z 385.987,A -85,B 0,C 180,E1 -11657.435,E2 -11657.435} C_VEL
LIN {X 0,Y 411.881,Z 386.988,A -85,B 0,C 180,E1 -11657.687,E2 -11657.687} C_VEL
LIN {X 0,Y 410.876,Z 391.512,A -85,B 0,C 180,E1 -11657.983,E2 -11657.983} C_VEL
LIN {X 0,Y 395.678,Z 460.676,A -85,B 0,C 180,E1 -11660.401,E2 -11660.401} C_VEL
LIN {X 0,Y 384.652,Z 522.343,A -85,B 0,C 180,E1 -11662.637,E2 -11662.637} C_VEL
LIN {X 0,Y 377.025,Z 574.21,A -85,B 0,C 180,E1 -11664.553,E2 -11664.553} C_VEL
LIN {X 0,Y 373.634,Z 595.093,A -85,B 0,C 180,E1 -11665.623,E2 -11665.623} C_VEL
LIN {X 0,Y 369.925,Z 615.815,A -85,B 0,C 180,E1 -11667.001,E2 -11667.001} C_VEL
LIN {X 0,Y 366.124,Z 635.487,A -85,B 0,C 180,E1 -11668.652,E2 -11668.652} C_VEL
LIN {X 0,Y 362.315,Z 654.128,A -85,B 0,C 180,E1 -11670.58,E2 -11670.58} C_VEL
LIN {X 0,Y 358.85,Z 670.387,A -85,B 0,C 180,E1 -11672.63,E2 -11672.63} C_VEL
LIN {X 0,Y 355.516,Z 685.664,A -85,B 0,C 180,E1 -11674.959,E2 -11674.959} C_VEL
LIN {X 0,Y 352.515,Z 699.304,A -85,B 0,C 180,E1 -11677.487,E2 -11677.487} C_VEL
LIN {X 0,Y 349.988,Z 710.975,A -85,B 0,C 180,E1 -11680.126,E2 -11680.126} C_VEL
LIN {X 0,Y 347.892,Z 721.126,A -85,B 0,C 180,E1 -11682.954,E2 -11682.954} C_VEL
LIN {X 0,Y 346.356,Z 729.292,A -85,B 0,C 180,E1 -11685.796,E2 -11685.796} C_VEL
LIN {X 0,Y 345.258,Z 735.992,A -85,B 0,C 180,E1 -11688.812,E2 -11688.812} C_VEL
LIN {X 0,Y 344.6,Z 740.879,A -85,B 0,C 180,E1 -11691.827,E2 -11691.827} C_VEL
LIN {X 0,Y 344.253,Z 744.174,A -85,B 0,C 180,E1 -11695.002,E2 -11695.002} C_VEL
LIN {X 0,Y 344.12,Z 745.622,A -85,B 0,C 180,E1 -11698.002,E2 -11698.002} C_VEL
LIN {X 0,Y 344.09,Z 745.431,A -85,B 0,C 180,E1 -11701,E2 -11701} C_VEL
LIN {X 0,Y 344.109,Z 743.619,A -85,B 0,C 180,E1 -11703.999,E2 -11703.999} C_VEL
LIN {X 0,Y 344.264,Z 740.153,A -85,B 0,C 180,E1 -11707.007,E2 -11707.007} C_VEL
LIN {X 0,Y 344.659,Z 734.945,A -85,B 0,C 180,E1 -11710.025,E2 -11710.025} C_VEL
LIN {X 0,Y 345.34,Z 728.301,A -85,B 0,C 180,E1 -11712.882,E2 -11712.882} C_VEL
LIN {X 0,Y 346.434,Z 719.818,A -85,B 0,C 180,E1 -11715.742,E2 -11715.742} C_VEL
LIN {X 0,Y 347.954,Z 709.604,A -85,B 0,C 180,E1 -11718.507,E2 -11718.507} C_VEL
LIN {X 0,Y 349.858,Z 697.859,A -85,B 0,C 180,E1 -11721.107,E2 -11721.107} C_VEL
LIN {X 0,Y 351.998,Z 685.158,A -85,B 0,C 180,E1 -11723.436,E2 -11723.436} C_VEL
LIN {X 0,Y 354.456,Z 670.589,A -85,B 0,C 180,E1 -11725.659,E2 -11725.659} C_VEL
LIN {X 0,Y 357.092,Z 654.42,A -85,B 0,C 180,E1 -11727.698,E2 -11727.698} C_VEL
LIN {X 0,Y 359.73,Z 637.257,A -85,B 0,C 180,E1 -11729.471,E2 -11729.471} C_VEL
LIN {X 0,Y 362.248,Z 619.175,A -85,B 0,C 180,E1 -11730.983,E2 -11730.983} C_VEL
LIN {X 0,Y 364.563,Z 599.974,A -85,B 0,C 180,E1 -11732.248,E2 -11732.248} C_VEL
LIN {X 0,Y 366.567,Z 579.862,A -85,B 0,C 180,E1 -11733.248,E2 -11733.248} C_VEL
LIN {X 0,Y 368.1,Z 559.726,A -85,B 0,C 180,E1 -11733.955,E2 -11733.955} C_VEL
LIN {X 0,Y 377.641,Z 380.802,A -85,B 0,C 180,E1 -11738.364,E2 -11738.364} C_VEL
LIN {X 0,Y 374.683,Z 359.244,A -85,B 0,C 180,E1 -11739.355,E2 -11739.355} C_VEL
LIN {X 0,Y 363.805,Z 338.545,A -85,B 0,C 180,E1 -11741.323,E2 -11741.323} C_VEL
LIN {X 0,Y 356.684,Z 319.845,A -85,B 0,C 180,E1 -11744.828,E2 -11744.828} C_VEL
LIN {X 0,Y 350.22,Z 304.007,A -85,B 0,C 180,E1 -11748.081,E2 -11748.081} C_VEL
LIN {X 0,Y 345.957,Z 293.592,A -85,B 0,C 180,E1 -11750.42,E2 -11750.42} C_VEL
LIN {X 0,Y 345.924,Z 293.396,A -85,B 0,C 180,E1 -11754.683,E2 -11754.683} C_VEL
LIN {X 0,Y 345.917,Z 293.39,A -85,B 0,C 180,E1 -11758.841,E2 -11758.841} C_VEL
LIN {X 0,Y 345.907,Z 293.399,A -85,B 0,C 180,E1 -11763.01,E2 -11763.01} C_VEL
LIN {X 0,Y 345.959,Z 293.599,A -85,B 0,C 180,E1 -11765.86,E2 -11765.86} C_VEL
LIN {X 0,Y 346.386,Z 295.233,A -85,B 0,C 180,E1 -11766.212,E2 -11766.212} C_VEL
LIN {X 0,Y 351.277,Z 305.801,A -85,B 0,C 180,E1 -11768.114,E2 -11768.114} C_VEL
LIN {X 0,Y 358.505,Z 323.211,A -85,B 0,C 180,E1 -11770.992,E2 -11770.992} C_VEL
LIN {X 0,Y 364.738,Z 340.658,A -85,B 0,C 180,E1 -11773.632,E2 -11773.632} C_VEL
LIN {X 0,Y 367.575,Z 349.984,A -85,B 0,C 180,E1 -11774.943,E2 -11774.943} C_VEL
LIN {X 0,Y 364.449,Z 392.246,A -85,B 0,C 180,E1 -11779.086,E2 -11779.086} C_VEL
LIN {X 0,Y 361.378,Z 433.081,A -85,B 0,C 180,E1 -11783.086,E2 -11783.086} C_VEL
LIN {X 0,Y 358.449,Z 474.145,A -85,B 0,C 180,E1 -11787.12,E2 -11787.12} C_VEL
LIN {X 0,Y 358.077,Z 481.347,A -85,B 0,C 180,E1 -11787.774,E2 -11787.774} C_VEL
LIN {X 0,Y 359.22,Z 491.389,A -85,B 0,C 180,E1 -11788.089,E2 -11788.089} C_VEL
LIN {X 0,Y 359.056,Z 497.957,A -85,B 0,C 180,E1 -11788.223,E2 -11788.223} C_VEL
LIN {X 0,Y 356.653,Z 507.714,A -85,B 0,C 180,E1 -11788.255,E2 -11788.255} C_VEL
LIN {X 0,Y 352.824,Z 520.75,A -85,B 0,C 180,E1 -11788.252,E2 -11788.252} C_VEL
LIN {X 0,Y 352.141,Z 526.316,A -85,B 0,C 180,E1 -11788.325,E2 -11788.325} C_VEL
LIN {X 0,Y 349.599,Z 625.09,A -85,B 0,C 180,E1 -11790.408,E2 -11790.408} C_VEL
LIN {X 0,Y 348.789,Z 641.248,A -85,B 0,C 180,E1 -11791.05,E2 -11791.05} C_VEL
LIN {X 0,Y 347.603,Z 656.897,A -85,B 0,C 180,E1 -11791.976,E2 -11791.976} C_VEL
LIN {X 0,Y 346.15,Z 671.38,A -85,B 0,C 180,E1 -11793.144,E2 -11793.144} C_VEL
LIN {X 0,Y 344.413,Z 685.801,A -85,B 0,C 180,E1 -11794.661,E2 -11794.661} C_VEL
LIN {X 0,Y 342.68,Z 698.496,A -85,B 0,C 180,E1 -11796.364,E2 -11796.364} C_VEL
LIN {X 0,Y 340.907,Z 710.688,A -85,B 0,C 180,E1 -11798.431,E2 -11798.431} C_VEL
LIN {X 0,Y 339.442,Z 720.467,A -85,B 0,C 180,E1 -11800.521,E2 -11800.521} C_VEL
LIN {X 0,Y 338.122,Z 729.538,A -85,B 0,C 180,E1 -11802.985,E2 -11802.985} C_VEL
LIN {X 0,Y 337.19,Z 736.557,A -85,B 0,C 180,E1 -11805.48,E2 -11805.48} C_VEL
LIN {X 0,Y 336.572,Z 742.076,A -85,B 0,C 180,E1 -11808.173,E2 -11808.173} C_VEL
LIN {X 0,Y 336.275,Z 745.59,A -85,B 0,C 180,E1 -11810.719,E2 -11810.719} C_VEL
LIN {X 0,Y 336.147,Z 747.599,A -85,B 0,C 180,E1 -11813.487,E2 -11813.487} C_VEL
LIN {X 0,Y 336.151,Z 747.893,A -85,B 0,C 180,E1 -11816.305,E2 -11816.305} C_VEL
LIN {X 0,Y 336.277,Z 746.368,A -85,B 0,C 180,E1 -11819.053,E2 -11819.053} C_VEL
LIN {X 0,Y 336.636,Z 742.95,A -85,B 0,C 180,E1 -11821.914,E2 -11821.914} C_VEL
LIN {X 0,Y 337.256,Z 738.038,A -85,B 0,C 180,E1 -11824.493,E2 -11824.493} C_VEL
LIN {X 0,Y 338.268,Z 731.244,A -85,B 0,C 180,E1 -11827.081,E2 -11827.081} C_VEL
LIN {X 0,Y 339.608,Z 722.889,A -85,B 0,C 180,E1 -11829.487,E2 -11829.487} C_VEL
LIN {X 0,Y 341.323,Z 712.507,A -85,B 0,C 180,E1 -11831.816,E2 -11831.816} C_VEL
LIN {X 0,Y 343.099,Z 701.367,A -85,B 0,C 180,E1 -11833.784,E2 -11833.784} C_VEL
LIN {X 0,Y 345.017,Z 688.531,A -85,B 0,C 180,E1 -11835.589,E2 -11835.589} C_VEL
LIN {X 0,Y 346.793,Z 675.042,A -85,B 0,C 180,E1 -11837.078,E2 -11837.078} C_VEL
LIN {X 0,Y 348.486,Z 659.849,A -85,B 0,C 180,E1 -11838.368,E2 -11838.368} C_VEL
LIN {X 0,Y 349.777,Z 644.4,A -85,B 0,C 180,E1 -11839.331,E2 -11839.331} C_VEL
LIN {X 0,Y 350.718,Z 627.649,A -85,B 0,C 180,E1 -11840.041,E2 -11840.041} C_VEL
LIN {X 0,Y 351.621,Z 594.862,A -85,B 0,C 180,E1 -11840.786,E2 -11840.786} C_VEL
LIN {X 0,Y 354.151,Z 499.226,A -85,B 0,C 180,E1 -11842.801,E2 -11842.801} C_VEL
LIN {X 0,Y 352.226,Z 481.476,A -85,B 0,C 180,E1 -11843.447,E2 -11843.447} C_VEL
LIN {X 0,Y 355.443,Z 439.199,A -85,B 0,C 180,E1 -11847.596,E2 -11847.596} C_VEL
LIN {X 0,Y 358.764,Z 397.06,A -85,B 0,C 180,E1 -11851.719,E2 -11851.719} C_VEL
LIN {X 0,Y 361.791,Z 356.157,A -85,B 0,C 180,E1 -11855.682,E2 -11855.682} C_VEL
LIN {X 0,Y 361.858,Z 351.927,A -85,B 0,C 180,E1 -11856.121,E2 -11856.121} C_VEL
LIN {X 0,Y 356.589,Z 335.585,A -85,B 0,C 180,E1 -11858.622,E2 -11858.622} C_VEL
LIN {X 0,Y 350.621,Z 320.641,A -85,B 0,C 180,E1 -11861.201,E2 -11861.201} C_VEL
LIN {X 0,Y 344.779,Z 307.854,A -85,B 0,C 180,E1 -11863.662,E2 -11863.662} C_VEL
LIN {X 0,Y 339.802,Z 298.575,A -85,B 0,C 180,E1 -11865.689,E2 -11865.689} C_VEL
LIN {X 0,Y 338.114,Z 295.101,A -85,B 0,C 180,E1 -11866.489,E2 -11866.489} C_VEL
LIN {X 0,Y 337.989,Z 294.413,A -85,B 0,C 180,E1 -11866.833,E2 -11866.833} C_VEL
LIN {X 0,Y 337.971,Z 294.384,A -85,B 0,C 180,E1 -11871.15,E2 -11871.15} C_VEL
LIN {X 0,Y 337.964,Z 294.384,A -85,B 0,C 180,E1 -11875.418,E2 -11875.418} C_VEL
LIN {X 0,Y 337.962,Z 294.388,A -85,B 0,C 180,E1 -11879.83,E2 -11879.83} C_VEL
LIN {X 0,Y 337.964,Z 294.38,A -85,B 0,C 180,E1 -11884.071,E2 -11884.071} C_VEL
LIN {X 0,Y 337.974,Z 294.388,A -85,B 0,C 180,E1 -11888.334,E2 -11888.334} C_VEL
LIN {X 0,Y 337.985,Z 294.377,A -85,B 0,C 180,E1 -11892.645,E2 -11892.645} C_VEL
LIN {X 0,Y 337.991,Z 294.382,A -85,B 0,C 180,E1 -11896.852,E2 -11896.852} C_VEL
LIN {X 0,Y 337.991,Z 294.379,A -85,B 0,C 180,E1 -11901.155,E2 -11901.155} C_VEL
LIN {X 0,Y 337.98,Z 294.382,A -85,B 0,C 180,E1 -11905.401,E2 -11905.401} C_VEL
LIN {X 0,Y 337.975,Z 294.381,A -85,B 0,C 180,E1 -11909.606,E2 -11909.606} C_VEL
LIN {X 0,Y 337.972,Z 294.383,A -85,B 0,C 180,E1 -11913.791,E2 -11913.791} C_VEL
LIN {X 0,Y 338.024,Z 294.627,A -85,B 0,C 180,E1 -11915.225,E2 -11915.225} C_VEL
LIN {X 0,Y 340.974,Z 301.625,A -85,B 0,C 180,E1 -11916.823,E2 -11916.823} C_VEL
LIN {X 0,Y 348.1,Z 317.658,A -85,B 0,C 180,E1 -11920.182,E2 -11920.182} C_VEL
LIN {X 0,Y 349.811,Z 321.321,A -85,B 0,C 180,E1 -11920.831,E2 -11920.831} C_VEL
LIN {X 0,Y 364.926,Z 347.052,A -85,B 0,C 180,E1 -11923.693,E2 -11923.693} C_VEL
LIN {X 0,Y 376.628,Z 368.263,A -85,B 0,C 180,E1 -11925.748,E2 -11925.748} C_VEL
LIN {X 0,Y 364.998,Z 577.035,A -85,B 0,C 180,E1 -11930.8,E2 -11930.8} C_VEL
LIN {X 0,Y 363.082,Z 598.522,A -85,B 0,C 180,E1 -11931.596,E2 -11931.596} C_VEL
LIN {X 0,Y 360.736,Z 618.858,A -85,B 0,C 180,E1 -11932.629,E2 -11932.629} C_VEL
LIN {X 0,Y 357.939,Z 639.326,A -85,B 0,C 180,E1 -11933.987,E2 -11933.987} C_VEL
LIN {X 0,Y 354.853,Z 659.156,A -85,B 0,C 180,E1 -11935.646,E2 -11935.646} C_VEL
LIN {X 0,Y 351.544,Z 678.422,A -85,B 0,C 180,E1 -11937.642,E2 -11937.642} C_VEL
LIN {X 0,Y 348.361,Z 695.927,A -85,B 0,C 180,E1 -11939.851,E2 -11939.851} C_VEL
LIN {X 0,Y 345.347,Z 712.086,A -85,B 0,C 180,E1 -11942.313,E2 -11942.313} C_VEL
LIN {X 0,Y 342.668,Z 726.607,A -85,B 0,C 180,E1 -11944.973,E2 -11944.973} C_VEL
LIN {X 0,Y 340.328,Z 739.902,A -85,B 0,C 180,E1 -11947.913,E2 -11947.913} C_VEL
LIN {X 0,Y 338.498,Z 751.508,A -85,B 0,C 180,E1 -11951.042,E2 -11951.042} C_VEL
LIN {X 0,Y 337.256,Z 760.909,A -85,B 0,C 180,E1 -11954.174,E2 -11954.174} C_VEL
LIN {X 0,Y 336.506,Z 768.386,A -85,B 0,C 180,E1 -11957.3,E2 -11957.3} C_VEL
LIN {X 0,Y 336.14,Z 774.404,A -85,B 0,C 180,E1 -11960.586,E2 -11960.586} C_VEL
LIN {X 0,Y 336.06,Z 778.451,A -85,B 0,C 180,E1 -11963.682,E2 -11963.682} C_VEL
LIN {X 0,Y 336.071,Z 780.929,A -85,B 0,C 180,E1 -11966.761,E2 -11966.761} C_VEL
LIN {X 0,Y 336.104,Z 781.831,A -85,B 0,C 180,E1 -11969.831,E2 -11969.831} C_VEL
LIN {X 0,Y 336.064,Z 781.192,A -85,B 0,C 180,E1 -11973.072,E2 -11973.072} C_VEL
LIN {X 0,Y 336.04,Z 779.085,A -85,B 0,C 180,E1 -11976.151,E2 -11976.151} C_VEL
LIN {X 0,Y 336.123,Z 775.131,A -85,B 0,C 180,E1 -11979.418,E2 -11979.418} C_VEL
LIN {X 0,Y 336.501,Z 769.44,A -85,B 0,C 180,E1 -11982.704,E2 -11982.704} C_VEL
LIN {X 0,Y 337.345,Z 761.904,A -85,B 0,C 180,E1 -11986.002,E2 -11986.002} C_VEL
LIN {X 0,Y 338.672,Z 752.894,A -85,B 0,C 180,E1 -11989.139,E2 -11989.139} C_VEL
LIN {X 0,Y 340.502,Z 742.618,A -85,B 0,C 180,E1 -11992.079,E2 -11992.079} C_VEL
LIN {X 0,Y 342.955,Z 730.241,A -85,B 0,C 180,E1 -11995.009,E2 -11995.009} C_VEL
LIN {X 0,Y 346.083,Z 715.492,A -85,B 0,C 180,E1 -11997.908,E2 -11997.908} C_VEL
LIN {X 0,Y 349.707,Z 698.984,A -85,B 0,C 180,E1 -12000.594,E2 -12000.594} C_VEL
LIN {X 0,Y 353.621,Z 681.141,A -85,B 0,C 180,E1 -12003,E2 -12003} C_VEL
LIN {X 0,Y 357.655,Z 662.442,A -85,B 0,C 180,E1 -12005.088,E2 -12005.088} C_VEL
LIN {X 0,Y 361.835,Z 642.249,A -85,B 0,C 180,E1 -12006.944,E2 -12006.944} C_VEL
LIN {X 0,Y 366.004,Z 621.018,A -85,B 0,C 180,E1 -12008.527,E2 -12008.527} C_VEL
LIN {X 0,Y 370.038,Z 599.043,A -85,B 0,C 180,E1 -12009.822,E2 -12009.822} C_VEL
LIN {X 0,Y 373.917,Z 575.802,A -85,B 0,C 180,E1 -12010.862,E2 -12010.862} C_VEL
LIN {X 0,Y 383.569,Z 511.855,A -85,B 0,C 180,E1 -12013.077,E2 -12013.077} C_VEL
LIN {X 0,Y 393.837,Z 459.479,A -85,B 0,C 180,E1 -12014.932,E2 -12014.932} C_VEL
LIN {X 0,Y 407.154,Z 404.303,A -85,B 0,C 180,E1 -12016.846,E2 -12016.846} C_VEL
LIN {X 0,Y 408.739,Z 398.253,A -85,B 0,C 180,E1 -12017.066,E2 -12017.066} C_VEL
LIN {X 0,Y 392.321,Z 466.817,A -85,B 0,C 180,E1 -12019.48,E2 -12019.48} C_VEL
LIN {X 0,Y 380.562,Z 526.134,A -85,B 0,C 180,E1 -12021.681,E2 -12021.681} C_VEL
LIN {X 0,Y 372.421,Z 575.002,A -85,B 0,C 180,E1 -12023.559,E2 -12023.559} C_VEL
LIN {X 0,Y 368.501,Z 596.344,A -85,B 0,C 180,E1 -12024.695,E2 -12024.695} C_VEL
LIN {X 0,Y 364.502,Z 616.293,A -85,B 0,C 180,E1 -12026.068,E2 -12026.068} C_VEL
LIN {X 0,Y 360.215,Z 636.313,A -85,B 0,C 180,E1 -12027.796,E2 -12027.796} C_VEL
LIN {X 0,Y 355.961,Z 655.265,A -85,B 0,C 180,E1 -12029.816,E2 -12029.816} C_VEL
LIN {X 0,Y 352.113,Z 671.811,A -85,B 0,C 180,E1 -12031.969,E2 -12031.969} C_VEL
LIN {X 0,Y 348.545,Z 686.8,A -85,B 0,C 180,E1 -12034.332,E2 -12034.332} C_VEL
LIN {X 0,Y 345.219,Z 700.605,A -85,B 0,C 180,E1 -12036.984,E2 -12036.984} C_VEL
LIN {X 0,Y 342.512,Z 712.08,A -85,B 0,C 180,E1 -12039.673,E2 -12039.673} C_VEL
LIN {X 0,Y 340.26,Z 722.087,A -85,B 0,C 180,E1 -12042.559,E2 -12042.559} C_VEL
LIN {X 0,Y 338.593,Z 730.136,A -85,B 0,C 180,E1 -12045.464,E2 -12045.464} C_VEL
LIN {X 0,Y 337.395,Z 736.734,A -85,B 0,C 180,E1 -12048.548,E2 -12048.548} C_VEL
LIN {X 0,Y 336.673,Z 741.533,A -85,B 0,C 180,E1 -12051.633,E2 -12051.633} C_VEL
LIN {X 0,Y 336.303,Z 744.635,A -85,B 0,C 180,E1 -12054.712,E2 -12054.712} C_VEL
LIN {X 0,Y 336.142,Z 746.084,A -85,B 0,C 180,E1 -12057.785,E2 -12057.785} C_VEL
LIN {X 0,Y 336.101,Z 745.899,A -85,B 0,C 180,E1 -12060.853,E2 -12060.853} C_VEL
LIN {X 0,Y 336.118,Z 744.091,A -85,B 0,C 180,E1 -12063.924,E2 -12063.924} C_VEL
LIN {X 0,Y 336.274,Z 740.622,A -85,B 0,C 180,E1 -12067.003,E2 -12067.003} C_VEL
LIN {X 0,Y 336.682,Z 735.404,A -85,B 0,C 180,E1 -12070.092,E2 -12070.092} C_VEL
LIN {X 0,Y 337.391,Z 728.745,A -85,B 0,C 180,E1 -12073.017,E2 -12073.017} C_VEL
LIN {X 0,Y 338.53,Z 720.238,A -85,B 0,C 180,E1 -12075.944,E2 -12075.944} C_VEL
LIN {X 0,Y 340.144,Z 709.81,A -85,B 0,C 180,E1 -12078.819,E2 -12078.819} C_VEL
LIN {X 0,Y 342.094,Z 698.219,A -85,B 0,C 180,E1 -12081.43,E2 -12081.43} C_VEL
LIN {X 0,Y 344.355,Z 685.278,A -85,B 0,C 180,E1 -12083.845,E2 -12083.845} C_VEL
LIN {X 0,Y 346.975,Z 670.305,A -85,B 0,C 180,E1 -12086.162,E2 -12086.162} C_VEL
LIN {X 0,Y 349.725,Z 653.999,A -85,B 0,C 180,E1 -12088.241,E2 -12088.241} C_VEL
LIN {X 0,Y 352.47,Z 636.673,A -85,B 0,C 180,E1 -12090.046,E2 -12090.046} C_VEL
LIN {X 0,Y 355.169,Z 617.678,A -85,B 0,C 180,E1 -12091.633,E2 -12091.633} C_VEL
LIN {X 0,Y 357.551,Z 598.311,A -85,B 0,C 180,E1 -12092.903,E2 -12092.903} C_VEL
LIN {X 0,Y 359.582,Z 578.331,A -85,B 0,C 180,E1 -12093.891,E2 -12093.891} C_VEL
LIN {X 0,Y 361.197,Z 557.274,A -85,B 0,C 180,E1 -12094.617,E2 -12094.617} C_VEL
LIN {X 0,Y 371.023,Z 381.928,A -85,B 0,C 180,E1 -12099.045,E2 -12099.045} C_VEL
LIN {X 0,Y 368.342,Z 362.58,A -85,B 0,C 180,E1 -12099.957,E2 -12099.957} C_VEL
LIN {X 0,Y 355.537,Z 338.327,A -85,B 0,C 180,E1 -12102.359,E2 -12102.359} C_VEL
LIN {X 0,Y 348.076,Z 318.918,A -85,B 0,C 180,E1 -12106.139,E2 -12106.139} C_VEL
LIN {X 0,Y 340.999,Z 301.781,A -85,B 0,C 180,E1 -12109.827,E2 -12109.827} C_VEL
LIN {X 0,Y 338.021,Z 294.573,A -85,B 0,C 180,E1 -12111.538,E2 -12111.538} C_VEL
LIN {X 0,Y 337.992,Z 294.383,A -85,B 0,C 180,E1 -12115.926,E2 -12115.926} C_VEL
LIN {X 0,Y 337.995,Z 294.356,A -85,B 0,C 180,E1 -12120.198,E2 -12120.198} C_VEL
LIN {X 0,Y 337.978,Z 294.364,A -85,B 0,C 180,E1 -12124.464,E2 -12124.464} C_VEL
LIN {X 0,Y 338.035,Z 294.816,A -85,B 0,C 180,E1 -12124.882,E2 -12124.882} C_VEL
LIN {X 0,Y 339.459,Z 298.103,A -85,B 0,C 180,E1 -12125.527,E2 -12125.527} C_VEL
LIN {X 0,Y 346.624,Z 313.982,A -85,B 0,C 180,E1 -12128.411,E2 -12128.411} C_VEL
LIN {X 0,Y 353.778,Z 331.98,A -85,B 0,C 180,E1 -12131.374,E2 -12131.374} C_VEL
LIN {X 0,Y 359.704,Z 349.633,A -85,B 0,C 180,E1 -12134.025,E2 -12134.025} C_VEL
LIN {X 0,Y 360.6,Z 352.898,A -85,B 0,C 180,E1 -12134.479,E2 -12134.479} C_VEL
LIN {X 0,Y 357.417,Z 393.918,A -85,B 0,C 180,E1 -12138.542,E2 -12138.542} C_VEL
LIN {X 0,Y 354.17,Z 435.046,A -85,B 0,C 180,E1 -12142.618,E2 -12142.618} C_VEL
LIN {X 0,Y 351.013,Z 477.267,A -85,B 0,C 180,E1 -12146.814,E2 -12146.814} C_VEL
LIN {X 0,Y 350.845,Z 481.781,A -85,B 0,C 180,E1 -12147.201,E2 -12147.201} C_VEL
LIN {X 0,Y 352.802,Z 501.673,A -85,B 0,C 180,E1 -12147.816,E2 -12147.816} C_VEL
LIN {X 0,Y 352.141,Z 526.316,A -85,B 0,C 180,E1 -12148.325,E2 -12148.325} C_VEL
LIN {X 0,Y 351.015,Z 533.985,A -85,B 0,C 180,E1 -12148.411,E2 -12148.411} C_VEL
LIN {X 0,Y 344.857,Z 554.319,A -85,B 0,C 180,E1 -12148.393,E2 -12148.393} C_VEL
LIN {X 0,Y 344.007,Z 560.903,A -85,B 0,C 180,E1 -12148.478,E2 -12148.478} C_VEL
LIN {X 0,Y 342.252,Z 625.857,A -85,B 0,C 180,E1 -12149.894,E2 -12149.894} C_VEL
LIN {X 0,Y 341.382,Z 642.145,A -85,B 0,C 180,E1 -12150.564,E2 -12150.564} C_VEL
LIN {X 0,Y 340.083,Z 658.406,A -85,B 0,C 180,E1 -12151.56,E2 -12151.56} C_VEL
LIN {X 0,Y 338.416,Z 673.874,A -85,B 0,C 180,E1 -12152.877,E2 -12152.877} C_VEL
LIN {X 0,Y 336.627,Z 687.872,A -85,B 0,C 180,E1 -12154.427,E2 -12154.427} C_VEL
LIN {X 0,Y 334.761,Z 700.769,A -85,B 0,C 180,E1 -12156.257,E2 -12156.257} C_VEL
LIN {X 0,Y 333.014,Z 712.162,A -85,B 0,C 180,E1 -12158.284,E2 -12158.284} C_VEL
LIN {X 0,Y 331.394,Z 722.426,A -85,B 0,C 180,E1 -12160.603,E2 -12160.603} C_VEL
LIN {X 0,Y 330.153,Z 730.631,A -85,B 0,C 180,E1 -12162.948,E2 -12162.948} C_VEL
LIN {X 0,Y 329.155,Z 737.778,A -85,B 0,C 180,E1 -12165.645,E2 -12165.645} C_VEL
LIN {X 0,Y 328.566,Z 742.901,A -85,B 0,C 180,E1 -12168.294,E2 -12168.294} C_VEL
LIN {X 0,Y 328.257,Z 746.362,A -85,B 0,C 180,E1 -12171.062,E2 -12171.062} C_VEL
LIN {X 0,Y 328.15,Z 748.169,A -85,B 0,C 180,E1 -12173.922,E2 -12173.922} C_VEL
LIN {X 0,Y 328.166,Z 748.212,A -85,B 0,C 180,E1 -12176.605,E2 -12176.605} C_VEL
LIN {X 0,Y 328.335,Z 746.434,A -85,B 0,C 180,E1 -12179.557,E2 -12179.557} C_VEL
LIN {X 0,Y 328.737,Z 742.939,A -85,B 0,C 180,E1 -12182.362,E2 -12182.362} C_VEL
LIN {X 0,Y 329.516,Z 737.416,A -85,B 0,C 180,E1 -12185.203,E2 -12185.203} C_VEL
LIN {X 0,Y 330.577,Z 730.877,A -85,B 0,C 180,E1 -12187.656,E2 -12187.656} C_VEL
